KUKA KRL program: EPS_2_251806_MH56A_A_20260213065153.src

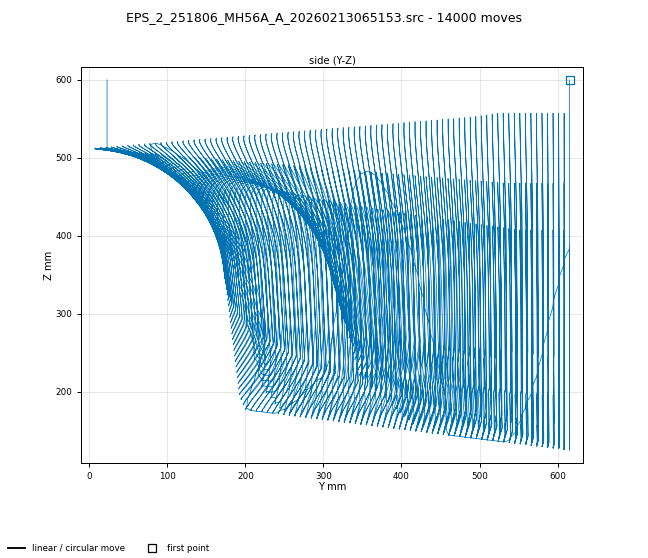
[picture p0: tool path of EPS_2_251806_MH56A_A_20260213065153.src, 14000 of 14002 moves have a stored position in this frame; points joined in program order, loops and branches not executed]
&ACCESS RVP
&REL 4
&COMMENT QRS 19112012
&PARAM EDITMASK = *
DEF PART()
EXT BAS (BAS_COMMAND :IN,REAL :IN )
INT I
BAS (#INITMOV,0 )

;KUKA QRS Post kuka4.cps  Date:22-06-2017 !

File_ID=3030

QRS_PRE_INIT()

;Init var - Until changes are made in qrs_pre_init
Outlet_Square_prg=0
Inlet_1_Square_prg=0
Inlet_2_Square_prg=0
Inlet_3_Square_prg=0
Inlet_4_Square_prg=0
Inlet_5_Square_prg=0

Outlet_1={X 0.000, Y 529.100, Z 408.000, B 0.000, E1 0.000 }
Inlet_1={X 0.000, Y 549.850, Z 257.000, B 0.000, E1 90.000 }
Inlet_2={X 0.000, Y 535.660, Z 318.000, B 0.000, E1 180.000 }
Outlet_1_type=299
Inlet_1_type=201
Inlet_2_type=299
;QRS#1=Sidecore dimensions
;QRS#2=300-12" PVC SDR 35
;QRS#3=200-8" PVC SDR 35
;QRS#4=300-12" PVC SDR 35
;QRS#5=
;QRS#6=
;QRS#7=
;QRS#8=
;QRS#9=16M PSX
;QRS#10=12-08 PSX
;QRS#11=16M PSX
;QRS#12=
;QRS#13=
;QRS#14=
;QRS#15=
;QRS#16=1220x127x838 2,75'
;QRS#17=EPS Height
;QRS#18=557,5
;QRS#19=*
;QRS#20= UPDATED VERSION 22-06-2017
;QRS#21=*
Outlet_Square=0150
Inlet_1_Square=0100
Inlet_2_Square=0150
Inlet_3_Square=0
Inlet_4_Square=0
Inlet_5_Square=0
Mill_Square=1
Outlet_Square_Prg=206
Inlet_1_Square_prg=204
Inlet_2_Square_prg=206

QRS_INIT()

$ADVANCE=5

; T1
PTP {E1 173.498,E2 173.498}
PTP {X 0,Y 615.498,A -85,B 0,C 180,E1 173.498,E2 173.498,E3 0,E4 0,E5 0,E6 0}
QRS_SPEED_INIT()
LIN {X 0,Y 615.498,Z 600,A -85,B 0,C 180,E1 173.498,E2 173.498,E3 0,E4 0,E5 0,E6 0} C_VEL
LIN {X 0,Y 615.498,Z 398.232,A -85,B 0,C 180,E1 173.498,E2 173.498} C_VEL
LIN {X 0,Y 615.498,Z 387.353,A -85,B 0,C 180,E1 173.498,E2 173.498} C_VEL
LIN {X 0,Y 615.496,Z 385.709,A -85,B 0,C 180,E1 173.418,E2 173.418} C_VEL
LIN {X 0,Y 615.498,Z 378.036,A -85,B 0,C 180,E1 172.455,E2 172.455} C_VEL
LIN {X 0,Y 615.498,Z 368.258,A -85,B 0,C 180,E1 171.463,E2 171.463} C_VEL
LIN {X 0,Y 615.497,Z 357.992,A -85,B 0,C 180,E1 170.636,E2 170.636} C_VEL
LIN {X 0,Y 615.487,Z 346.429,A -85,B 0,C 180,E1 169.889,E2 169.889} C_VEL
LIN {X 0,Y 615.498,Z 334.597,A -85,B 0,C 180,E1 169.294,E2 169.294} C_VEL
LIN {X 0,Y 615.462,Z 321.661,A -85,B 0,C 180,E1 168.806,E2 168.806} C_VEL
LIN {X 0,Y 615.456,Z 309.061,A -85,B 0,C 180,E1 168.473,E2 168.473} C_VEL
LIN {X 0,Y 615.464,Z 295.936,A -85,B 0,C 180,E1 168.264,E2 168.264} C_VEL
LIN {X 0,Y 615.464,Z 195.1,A -85,B 0,C 180,E1 167.071,E2 167.071} C_VEL
LIN {X 0,Y 615.457,Z 175.283,A -85,B 0,C 180,E1 164.434,E2 164.434} C_VEL
LIN {X 0,Y 615.488,Z 153.929,A -85,B 0,C 180,E1 161.558,E2 161.558} C_VEL
LIN {X 0,Y 615.464,Z 133.353,A -85,B 0,C 180,E1 158.743,E2 158.743} C_VEL
LIN {X 0,Y 615.471,Z 125.313,A -85,B 0,C 180,E1 157.627,E2 157.627} C_VEL
LIN {X 0,Y 615.452,Z 125.319,A -85,B 0,C 180,E1 155.007,E2 155.007} C_VEL
LIN {X 0,Y 615.489,Z 125.315,A -85,B 0,C 180,E1 152.085,E2 152.085} C_VEL
LIN {X 0,Y 615.481,Z 125.311,A -85,B 0,C 180,E1 149.839,E2 149.839} C_VEL
LIN {X 0,Y 615.458,Z 125.315,A -85,B 0,C 180,E1 147.541,E2 147.541} C_VEL
LIN {X 0,Y 615.459,Z 125.319,A -85,B 0,C 180,E1 145.183,E2 145.183} C_VEL
LIN {X 0,Y 615.488,Z 125.327,A -85,B 0,C 180,E1 142.758,E2 142.758} C_VEL
LIN {X 0,Y 615.475,Z 125.311,A -85,B 0,C 180,E1 139.913,E2 139.913} C_VEL
LIN {X 0,Y 615.461,Z 125.315,A -85,B 0,C 180,E1 137.645,E2 137.645} C_VEL
LIN {X 0,Y 615.495,Z 125.326,A -85,B 0,C 180,E1 134.932,E2 134.932} C_VEL
LIN {X 0,Y 615.479,Z 125.31,A -85,B 0,C 180,E1 132.079,E2 132.079} C_VEL
LIN {X 0,Y 615.464,Z 125.315,A -85,B 0,C 180,E1 129.753,E2 129.753} C_VEL
LIN {X 0,Y 615.487,Z 125.321,A -85,B 0,C 180,E1 126.936,E2 126.936} C_VEL
LIN {X 0,Y 615.469,Z 125.313,A -85,B 0,C 180,E1 124.024,E2 124.024} C_VEL
LIN {X 0,Y 615.468,Z 125.319,A -85,B 0,C 180,E1 121.687,E2 121.687} C_VEL
LIN {X 0,Y 615.486,Z 125.326,A -85,B 0,C 180,E1 119.407,E2 119.407} C_VEL
LIN {X 0,Y 615.485,Z 125.308,A -85,B 0,C 180,E1 116.445,E2 116.445} C_VEL
LIN {X 0,Y 615.485,Z 125.326,A -85,B 0,C 180,E1 113.557,E2 113.557} C_VEL
LIN {X 0,Y 615.476,Z 125.335,A -85,B 0,C 180,E1 112.266,E2 112.266} C_VEL
LIN {X 0,Y 615.46,Z 145.204,A -85,B 0,C 180,E1 109.687,E2 109.687} C_VEL
LIN {X 0,Y 615.464,Z 157.175,A -85,B 0,C 180,E1 108.18,E2 108.18} C_VEL
LIN {X 0,Y 615.492,Z 321.221,A -85,B 0,C 180,E1 106.201,E2 106.201} C_VEL
LIN {X 0,Y 615.489,Z 335.787,A -85,B 0,C 180,E1 105.906,E2 105.906} C_VEL
LIN {X 0,Y 615.477,Z 350.397,A -85,B 0,C 180,E1 105.481,E2 105.481} C_VEL
LIN {X 0,Y 615.492,Z 363.722,A -85,B 0,C 180,E1 104.973,E2 104.973} C_VEL
LIN {X 0,Y 615.483,Z 377.372,A -85,B 0,C 180,E1 104.32,E2 104.32} C_VEL
LIN {X 0,Y 615.5,Z 390.656,A -85,B 0,C 180,E1 103.538,E2 103.538} C_VEL
LIN {X 0,Y 615.497,Z 402.508,A -85,B 0,C 180,E1 102.698,E2 102.698} C_VEL
LIN {X 0,Y 615.497,Z 414.352,A -85,B 0,C 180,E1 101.694,E2 101.694} C_VEL
LIN {X 0,Y 615.495,Z 424.163,A -85,B 0,C 180,E1 100.709,E2 100.709} C_VEL
LIN {X 0,Y 615.495,Z 434.007,A -85,B 0,C 180,E1 99.531,E2 99.531} C_VEL
LIN {X 0,Y 615.497,Z 442.098,A -85,B 0,C 180,E1 98.372,E2 98.372} C_VEL
LIN {X 0,Y 615.491,Z 448.779,A -85,B 0,C 180,E1 97.216,E2 97.216} C_VEL
LIN {X 0,Y 615.499,Z 454.945,A -85,B 0,C 180,E1 95.899,E2 95.899} C_VEL
LIN {X 0,Y 615.489,Z 459.714,A -85,B 0,C 180,E1 94.585,E2 94.585} C_VEL
LIN {X 0,Y 615.491,Z 463.219,A -85,B 0,C 180,E1 93.274,E2 93.274} C_VEL
LIN {X 0,Y 615.5,Z 465.539,A -85,B 0,C 180,E1 91.964,E2 91.964} C_VEL
LIN {X 0,Y 615.491,Z 466.728,A -85,B 0,C 180,E1 90.655,E2 90.655} C_VEL
LIN {X 0,Y 615.492,Z 466.751,A -85,B 0,C 180,E1 89.347,E2 89.347} C_VEL
LIN {X 0,Y 615.5,Z 465.647,A -85,B 0,C 180,E1 88.038,E2 88.038} C_VEL
LIN {X 0,Y 615.494,Z 463.417,A -85,B 0,C 180,E1 86.728,E2 86.728} C_VEL
LIN {X 0,Y 615.49,Z 460.008,A -85,B 0,C 180,E1 85.416,E2 85.416} C_VEL
LIN {X 0,Y 615.499,Z 455.339,A -85,B 0,C 180,E1 84.102,E2 84.102} C_VEL
LIN {X 0,Y 615.491,Z 449.277,A -85,B 0,C 180,E1 82.785,E2 82.785} C_VEL
LIN {X 0,Y 615.493,Z 441.639,A -85,B 0,C 180,E1 81.464,E2 81.464} C_VEL
LIN {X 0,Y 615.496,Z 433.457,A -85,B 0,C 180,E1 80.305,E2 80.305} C_VEL
LIN {X 0,Y 615.495,Z 423.338,A -85,B 0,C 180,E1 79.109,E2 79.109} C_VEL
LIN {X 0,Y 615.497,Z 411.693,A -85,B 0,C 180,E1 77.973,E2 77.973} C_VEL
LIN {X 0,Y 615.498,Z 400.425,A -85,B 0,C 180,E1 77.052,E2 77.052} C_VEL
LIN {X 0,Y 615.498,Z 388.189,A -85,B 0,C 180,E1 76.211,E2 76.211} C_VEL
LIN {X 0,Y 615.49,Z 374.794,A -85,B 0,C 180,E1 75.452,E2 75.452} C_VEL
LIN {X 0,Y 615.488,Z 359.885,A -85,B 0,C 180,E1 74.775,E2 74.775} C_VEL
LIN {X 0,Y 615.476,Z 345.415,A -85,B 0,C 180,E1 74.266,E2 74.266} C_VEL
LIN {X 0,Y 615.492,Z 329.776,A -85,B 0,C 180,E1 73.865,E2 73.865} C_VEL
LIN {X 0,Y 615.492,Z 314.76,A -85,B 0,C 180,E1 73.618,E2 73.618} C_VEL
LIN {X 0,Y 615.47,Z 156.862,A -85,B 0,C 180,E1 71.72,E2 71.72} C_VEL
LIN {X 0,Y 615.478,Z 135.121,A -85,B 0,C 180,E1 68.92,E2 68.92} C_VEL
LIN {X 0,Y 615.483,Z 125.31,A -85,B 0,C 180,E1 67.625,E2 67.625} C_VEL
LIN {X 0,Y 615.478,Z 125.313,A -85,B 0,C 180,E1 65.009,E2 65.009} C_VEL
LIN {X 0,Y 615.476,Z 125.318,A -85,B 0,C 180,E1 62.823,E2 62.823} C_VEL
LIN {X 0,Y 615.482,Z 125.319,A -85,B 0,C 180,E1 60.207,E2 60.207} C_VEL
LIN {X 0,Y 615.493,Z 125.306,A -85,B 0,C 180,E1 57.544,E2 57.544} C_VEL
LIN {X 0,Y 615.477,Z 125.312,A -85,B 0,C 180,E1 55.186,E2 55.186} C_VEL
LIN {X 0,Y 615.486,Z 125.322,A -85,B 0,C 180,E1 52.759,E2 52.759} C_VEL
LIN {X 0,Y 615.482,Z 125.31,A -85,B 0,C 180,E1 49.912,E2 49.912} C_VEL
LIN {X 0,Y 615.495,Z 125.306,A -85,B 0,C 180,E1 47.649,E2 47.649} C_VEL
LIN {X 0,Y 615.478,Z 125.321,A -85,B 0,C 180,E1 44.932,E2 44.932} C_VEL
LIN {X 0,Y 615.483,Z 125.311,A -85,B 0,C 180,E1 42.082,E2 42.082} C_VEL
LIN {X 0,Y 615.489,Z 125.307,A -85,B 0,C 180,E1 39.75,E2 39.75} C_VEL
LIN {X 0,Y 615.482,Z 125.324,A -85,B 0,C 180,E1 36.938,E2 36.938} C_VEL
LIN {X 0,Y 615.488,Z 125.308,A -85,B 0,C 180,E1 34.022,E2 34.022} C_VEL
LIN {X 0,Y 615.479,Z 125.322,A -85,B 0,C 180,E1 31.087,E2 31.087} C_VEL
LIN {X 0,Y 615.482,Z 125.314,A -85,B 0,C 180,E1 28.452,E2 28.452} C_VEL
LIN {X 0,Y 615.476,Z 125.311,A -85,B 0,C 180,E1 25.716,E2 25.716} C_VEL
LIN {X 0,Y 615.472,Z 125.315,A -85,B 0,C 180,E1 23.557,E2 23.557} C_VEL
LIN {X 0,Y 615.473,Z 125.318,A -85,B 0,C 180,E1 21.433,E2 21.433} C_VEL
LIN {X 0,Y 615.483,Z 125.315,A -85,B 0,C 180,E1 18.608,E2 18.608} C_VEL
LIN {X 0,Y 615.476,Z 125.311,A -85,B 0,C 180,E1 15.906,E2 15.906} C_VEL
LIN {X 0,Y 615.49,Z 125.325,A -85,B 0,C 180,E1 13.201,E2 13.201} C_VEL
LIN {X 0,Y 615.488,Z 125.31,A -85,B 0,C 180,E1 10.527,E2 10.527} C_VEL
LIN {X 0,Y 615.47,Z 125.313,A -85,B 0,C 180,E1 7.876,E2 7.876} C_VEL
LIN {X 0,Y 615.493,Z 125.327,A -85,B 0,C 180,E1 5.241,E2 5.241} C_VEL
LIN {X 0,Y 615.491,Z 125.309,A -85,B 0,C 180,E1 2.618,E2 2.618} C_VEL
LIN {X 0,Y 615.469,Z 125.314,A -85,B 0,C 180,E1 0,E2 0} C_VEL
LIN {X 0,Y 615.489,Z 125.326,A -85,B 0,C 180,E1 -2.618,E2 -2.618} C_VEL
LIN {X 0,Y 615.491,Z 125.31,A -85,B 0,C 180,E1 -5.241,E2 -5.241} C_VEL
LIN {X 0,Y 615.467,Z 125.314,A -85,B 0,C 180,E1 -7.876,E2 -7.876} C_VEL
LIN {X 0,Y 615.489,Z 125.327,A -85,B 0,C 180,E1 -10.527,E2 -10.527} C_VEL
LIN {X 0,Y 615.495,Z 125.308,A -85,B 0,C 180,E1 -13.201,E2 -13.201} C_VEL
LIN {X 0,Y 615.465,Z 125.316,A -85,B 0,C 180,E1 -15.906,E2 -15.906} C_VEL
LIN {X 0,Y 615.49,Z 125.32,A -85,B 0,C 180,E1 -18.646,E2 -18.646} C_VEL
LIN {X 0,Y 615.475,Z 125.31,A -85,B 0,C 180,E1 -21.432,E2 -21.432} C_VEL
LIN {X 0,Y 615.486,Z 125.325,A -85,B 0,C 180,E1 -24.272,E2 -24.272} C_VEL
LIN {X 0,Y 615.487,Z 125.308,A -85,B 0,C 180,E1 -27.177,E2 -27.177} C_VEL
LIN {X 0,Y 615.465,Z 125.318,A -85,B 0,C 180,E1 -29.793,E2 -29.793} C_VEL
LIN {X 0,Y 615.49,Z 125.32,A -85,B 0,C 180,E1 -32.457,E2 -32.457} C_VEL
LIN {X 0,Y 615.493,Z 125.309,A -85,B 0,C 180,E1 -34.815,E2 -34.815} C_VEL
LIN {X 0,Y 615.469,Z 125.312,A -85,B 0,C 180,E1 -37.243,E2 -37.243} C_VEL
LIN {X 0,Y 615.494,Z 125.324,A -85,B 0,C 180,E1 -40.092,E2 -40.092} C_VEL
LIN {X 0,Y 615.474,Z 125.31,A -85,B 0,C 180,E1 -43.048,E2 -43.048} C_VEL
LIN {X 0,Y 615.478,Z 125.322,A -85,B 0,C 180,E1 -45.851,E2 -45.851} C_VEL
LIN {X 0,Y 615.493,Z 125.311,A -85,B 0,C 180,E1 -48.528,E2 -48.528} C_VEL
LIN {X 0,Y 615.464,Z 125.313,A -85,B 0,C 180,E1 -51.095,E2 -51.095} C_VEL
LIN {X 0,Y 615.466,Z 125.32,A -85,B 0,C 180,E1 -53.575,E2 -53.575} C_VEL
LIN {X 0,Y 615.495,Z 125.31,A -85,B 0,C 180,E1 -56.465,E2 -56.465} C_VEL
LIN {X 0,Y 615.459,Z 125.315,A -85,B 0,C 180,E1 -59.08,E2 -59.08} C_VEL
LIN {X 0,Y 615.471,Z 125.321,A -85,B 0,C 180,E1 -61.553,E2 -61.553} C_VEL
LIN {X 0,Y 615.473,Z 125.335,A -85,B 0,C 180,E1 -62.731,E2 -62.731} C_VEL
LIN {X 0,Y 615.474,Z 159.072,A -85,B 0,C 180,E1 -65.369,E2 -65.369} C_VEL
LIN {X 0,Y 615.491,Z 196.299,A -85,B 0,C 180,E1 -68.218,E2 -68.218} C_VEL
LIN {X 0,Y 615.474,Z 234.689,A -85,B 0,C 180,E1 -71.095,E2 -71.095} C_VEL
LIN {X 0,Y 615.483,Z 243.095,A -85,B 0,C 180,E1 -71.719,E2 -71.719} C_VEL
LIN {X 0,Y 615.482,Z 412.295,A -85,B 0,C 180,E1 -73.77,E2 -73.77} C_VEL
LIN {X 0,Y 615.496,Z 427.753,A -85,B 0,C 180,E1 -74.096,E2 -74.096} C_VEL
LIN {X 0,Y 615.481,Z 443.079,A -85,B 0,C 180,E1 -74.563,E2 -74.563} C_VEL
LIN {X 0,Y 615.497,Z 456.777,A -85,B 0,C 180,E1 -75.114,E2 -75.114} C_VEL
LIN {X 0,Y 615.495,Z 471.053,A -85,B 0,C 180,E1 -75.834,E2 -75.834} C_VEL
LIN {X 0,Y 615.497,Z 483.914,A -85,B 0,C 180,E1 -76.632,E2 -76.632} C_VEL
LIN {X 0,Y 615.495,Z 496.267,A -85,B 0,C 180,E1 -77.555,E2 -77.555} C_VEL
LIN {X 0,Y 615.495,Z 506.617,A -85,B 0,C 180,E1 -78.474,E2 -78.474} C_VEL
LIN {X 0,Y 615.495,Z 516.193,A -85,B 0,C 180,E1 -79.474,E2 -79.474} C_VEL
LIN {X 0,Y 615.493,Z 525.584,A -85,B 0,C 180,E1 -80.637,E2 -80.637} C_VEL
LIN {X 0,Y 615.494,Z 533.386,A -85,B 0,C 180,E1 -81.795,E2 -81.795} C_VEL
LIN {X 0,Y 615.496,Z 540.608,A -85,B 0,C 180,E1 -83.102,E2 -83.102} C_VEL
LIN {X 0,Y 615.499,Z 546.44,A -85,B 0,C 180,E1 -84.431,E2 -84.431} C_VEL
LIN {X 0,Y 615.491,Z 549.863,A -85,B 0,C 180,E1 -85.416,E2 -85.416} C_VEL
LIN {X 0,Y 615.492,Z 553.32,A -85,B 0,C 180,E1 -86.728,E2 -86.728} C_VEL
LIN {X 0,Y 615.499,Z 555.594,A -85,B 0,C 180,E1 -88.038,E2 -88.038} C_VEL
LIN {X 0,Y 615.494,Z 556.741,A -85,B 0,C 180,E1 -89.347,E2 -89.347} C_VEL
LIN {X 0,Y 615.494,Z 556.74,A -85,B 0,C 180,E1 -90.655,E2 -90.655} C_VEL
LIN {X 0,Y 615.499,Z 555.592,A -85,B 0,C 180,E1 -91.964,E2 -91.964} C_VEL
LIN {X 0,Y 615.492,Z 553.316,A -85,B 0,C 180,E1 -93.274,E2 -93.274} C_VEL
LIN {X 0,Y 615.491,Z 549.858,A -85,B 0,C 180,E1 -94.585,E2 -94.585} C_VEL
LIN {X 0,Y 615.499,Z 545.138,A -85,B 0,C 180,E1 -95.899,E2 -95.899} C_VEL
LIN {X 0,Y 615.494,Z 539.025,A -85,B 0,C 180,E1 -97.216,E2 -97.216} C_VEL
LIN {X 0,Y 615.494,Z 531.327,A -85,B 0,C 180,E1 -98.537,E2 -98.537} C_VEL
LIN {X 0,Y 615.495,Z 523.108,A -85,B 0,C 180,E1 -99.697,E2 -99.697} C_VEL
LIN {X 0,Y 615.497,Z 512.892,A -85,B 0,C 180,E1 -100.893,E2 -100.893} C_VEL
LIN {X 0,Y 615.495,Z 503.059,A -85,B 0,C 180,E1 -101.861,E2 -101.861} C_VEL
LIN {X 0,Y 615.497,Z 490.937,A -85,B 0,C 180,E1 -102.866,E2 -102.866} C_VEL
LIN {X 0,Y 615.498,Z 478.786,A -85,B 0,C 180,E1 -103.706,E2 -103.706} C_VEL
LIN {X 0,Y 615.488,Z 465.367,A -85,B 0,C 180,E1 -104.473,E2 -104.473} C_VEL
LIN {X 0,Y 615.497,Z 450.831,A -85,B 0,C 180,E1 -105.142,E2 -105.142} C_VEL
LIN {X 0,Y 615.495,Z 436.593,A -85,B 0,C 180,E1 -105.651,E2 -105.651} C_VEL
LIN {X 0,Y 615.498,Z 422.148,A -85,B 0,C 180,E1 -106.035,E2 -106.035} C_VEL
LIN {X 0,Y 615.479,Z 407.742,A -85,B 0,C 180,E1 -106.296,E2 -106.296} C_VEL
LIN {X 0,Y 615.483,Z 243.081,A -85,B 0,C 180,E1 -108.282,E2 -108.282} C_VEL
LIN {X 0,Y 615.495,Z 205.582,A -85,B 0,C 180,E1 -111.081,E2 -111.081} C_VEL
LIN {X 0,Y 615.487,Z 170.098,A -85,B 0,C 180,E1 -113.78,E2 -113.78} C_VEL
LIN {X 0,Y 615.473,Z 135.781,A -85,B 0,C 180,E1 -116.445,E2 -116.445} C_VEL
LIN {X 0,Y 615.47,Z 125.313,A -85,B 0,C 180,E1 -117.271,E2 -117.271} C_VEL
LIN {X 0,Y 615.483,Z 125.324,A -85,B 0,C 180,E1 -120.161,E2 -120.161} C_VEL
LIN {X 0,Y 615.45,Z 125.321,A -85,B 0,C 180,E1 -122.46,E2 -122.46} C_VEL
LIN {X 0,Y 615.447,Z 125.318,A -85,B 0,C 180,E1 -124.818,E2 -124.818} C_VEL
LIN {X 0,Y 615.477,Z 125.316,A -85,B 0,C 180,E1 -127.244,E2 -127.244} C_VEL
LIN {X 0,Y 615.446,Z 125.323,A -85,B 0,C 180,E1 -130.085,E2 -130.085} C_VEL
LIN {X 0,Y 615.43,Z 125.322,A -85,B 0,C 180,E1 -132.359,E2 -132.359} C_VEL
LIN {X 0,Y 615.457,Z 125.321,A -85,B 0,C 180,E1 -134.929,E2 -134.929} C_VEL
LIN {X 0,Y 615.451,Z 125.325,A -85,B 0,C 180,E1 -137.644,E2 -137.644} C_VEL
LIN {X 0,Y 615.415,Z 125.325,A -85,B 0,C 180,E1 -140.244,E2 -140.244} C_VEL
LIN {X 0,Y 615.455,Z 125.325,A -85,B 0,C 180,E1 -142.756,E2 -142.756} C_VEL
LIN {X 0,Y 615.468,Z 125.321,A -85,B 0,C 180,E1 -145.303,E2 -145.303} C_VEL
LIN {X 0,Y 615.432,Z 125.322,A -85,B 0,C 180,E1 -147.678,E2 -147.678} C_VEL
LIN {X 0,Y 615.431,Z 125.321,A -85,B 0,C 180,E1 -149.837,E2 -149.837} C_VEL
LIN {X 0,Y 615.441,Z 125.322,A -85,B 0,C 180,E1 -152.083,E2 -152.083} C_VEL
LIN {X 0,Y 615.477,Z 125.325,A -85,B 0,C 180,E1 -154.434,E2 -154.434} C_VEL
LIN {X 0,Y 615.469,Z 125.315,A -85,B 0,C 180,E1 -157.155,E2 -157.155} C_VEL
LIN {X 0,Y 615.446,Z 125.455,A -85,B 0,C 180,E1 -157.739,E2 -157.739} C_VEL
LIN {X 0,Y 615.475,Z 144.141,A -85,B 0,C 180,E1 -160.315,E2 -160.315} C_VEL
LIN {X 0,Y 615.474,Z 165.728,A -85,B 0,C 180,E1 -163.242,E2 -163.242} C_VEL
LIN {X 0,Y 615.456,Z 185.766,A -85,B 0,C 180,E1 -165.922,E2 -165.922} C_VEL
LIN {X 0,Y 615.467,Z 195.354,A -85,B 0,C 180,E1 -167.176,E2 -167.176} C_VEL
LIN {X 0,Y 615.489,Z 303.148,A -85,B 0,C 180,E1 -168.452,E2 -168.452} C_VEL
LIN {X 0,Y 615.494,Z 315.725,A -85,B 0,C 180,E1 -168.724,E2 -168.724} C_VEL
LIN {X 0,Y 615.493,Z 329.078,A -85,B 0,C 180,E1 -169.157,E2 -169.157} C_VEL
LIN {X 0,Y 615.47,Z 340.07,A -85,B 0,C 180,E1 -169.639,E2 -169.639} C_VEL
LIN {X 0,Y 615.47,Z 351.809,A -85,B 0,C 180,E1 -170.304,E2 -170.304} C_VEL
LIN {X 0,Y 615.499,Z 362.268,A -85,B 0,C 180,E1 -171.05,E2 -171.05} C_VEL
LIN {X 0,Y 615.498,Z 370.831,A -85,B 0,C 180,E1 -171.794,E2 -171.794} C_VEL
LIN {X 0,Y 615.497,Z 378.71,A -85,B 0,C 180,E1 -172.62,E2 -172.62} C_VEL
LIN {X 0,Y 615.497,Z 386.399,A -85,B 0,C 180,E1 -173.608,E2 -173.608} C_VEL
LIN {X 0,Y 615.497,Z 393.458,A -85,B 0,C 180,E1 -174.759,E2 -174.759} C_VEL
LIN {X 0,Y 615.497,Z 398.157,A -85,B 0,C 180,E1 -175.744,E2 -175.744} C_VEL
LIN {X 0,Y 615.495,Z 401.755,A -85,B 0,C 180,E1 -176.727,E2 -176.727} C_VEL
LIN {X 0,Y 615.496,Z 403.615,A -85,B 0,C 180,E1 -177.382,E2 -177.382} C_VEL
LIN {X 0,Y 615.497,Z 405.034,A -85,B 0,C 180,E1 -178.037,E2 -178.037} C_VEL
LIN {X 0,Y 615.497,Z 406.641,A -85,B 0,C 180,E1 -179.346,E2 -179.346} C_VEL
LIN {X 0,Y 615.494,Z 406.884,A -85,B 0,C 180,E1 -180,E2 -180} C_VEL
LIN {X 0,Y 615.495,Z 406.705,A -85,B 0,C 180,E1 -180.654,E2 -180.654} C_VEL
LIN {X 0,Y 615.496,Z 405.183,A -85,B 0,C 180,E1 -181.963,E2 -181.963} C_VEL
LIN {X 0,Y 615.498,Z 403.841,A -85,B 0,C 180,E1 -182.618,E2 -182.618} C_VEL
LIN {X 0,Y 615.497,Z 400.994,A -85,B 0,C 180,E1 -183.601,E2 -183.601} C_VEL
LIN {X 0,Y 615.498,Z 397.134,A -85,B 0,C 180,E1 -184.585,E2 -184.585} C_VEL
LIN {X 0,Y 615.498,Z 392.151,A -85,B 0,C 180,E1 -185.57,E2 -185.57} C_VEL
LIN {X 0,Y 615.496,Z 385.709,A -85,B 0,C 180,E1 -186.582,E2 -186.582} C_VEL
LIN {X 0,Y 614.829,Z 382.527,A -85,B 0,C 180,E1 -187.031,E2 -187.031} C_VEL
LIN {X 0,Y 611.989,Z 376.954,A -85,B 0,C 180,E1 -187.748,E2 -187.748} C_VEL
LIN {X 0,Y 609.138,Z 370.679,A -85,B 0,C 180,E1 -188.429,E2 -188.429} C_VEL
LIN {X 0,Y 608.477,Z 366.438,A -85,B 0,C 180,E1 -188.819,E2 -188.819} C_VEL
LIN {X 0,Y 608.491,Z 355.888,A -85,B 0,C 180,E1 -189.641,E2 -189.641} C_VEL
LIN {X 0,Y 608.492,Z 345.11,A -85,B 0,C 180,E1 -190.313,E2 -190.313} C_VEL
LIN {X 0,Y 608.518,Z 332.676,A -85,B 0,C 180,E1 -190.918,E2 -190.918} C_VEL
LIN {X 0,Y 608.496,Z 320.463,A -85,B 0,C 180,E1 -191.366,E2 -191.366} C_VEL
LIN {X 0,Y 608.528,Z 308.153,A -85,B 0,C 180,E1 -191.682,E2 -191.682} C_VEL
LIN {X 0,Y 608.54,Z 294.245,A -85,B 0,C 180,E1 -191.893,E2 -191.893} C_VEL
LIN {X 0,Y 608.511,Z 195.849,A -85,B 0,C 180,E1 -193.058,E2 -193.058} C_VEL
LIN {X 0,Y 608.45,Z 195.084,A -85,B 0,C 180,E1 -193.102,E2 -193.102} C_VEL
LIN {X 0,Y 608.469,Z 176.629,A -85,B 0,C 180,E1 -195.578,E2 -195.578} C_VEL
LIN {X 0,Y 608.533,Z 155.148,A -85,B 0,C 180,E1 -198.496,E2 -198.496} C_VEL
LIN {X 0,Y 608.55,Z 134.625,A -85,B 0,C 180,E1 -201.333,E2 -201.333} C_VEL
LIN {X 0,Y 608.458,Z 126.314,A -85,B 0,C 180,E1 -202.527,E2 -202.527} C_VEL
LIN {X 0,Y 608.438,Z 126.315,A -85,B 0,C 180,E1 -204.572,E2 -204.572} C_VEL
LIN {X 0,Y 608.461,Z 126.317,A -85,B 0,C 180,E1 -207.203,E2 -207.203} C_VEL
LIN {X 0,Y 608.471,Z 126.313,A -85,B 0,C 180,E1 -209.971,E2 -209.971} C_VEL
LIN {X 0,Y 608.448,Z 126.316,A -85,B 0,C 180,E1 -212.88,E2 -212.88} C_VEL
LIN {X 0,Y 608.437,Z 126.325,A -85,B 0,C 180,E1 -215.278,E2 -215.278} C_VEL
LIN {X 0,Y 608.466,Z 126.314,A -85,B 0,C 180,E1 -217.747,E2 -217.747} C_VEL
LIN {X 0,Y 608.437,Z 126.315,A -85,B 0,C 180,E1 -220.327,E2 -220.327} C_VEL
LIN {X 0,Y 608.481,Z 126.316,A -85,B 0,C 180,E1 -223.309,E2 -223.309} C_VEL
LIN {X 0,Y 608.461,Z 126.312,A -85,B 0,C 180,E1 -226.129,E2 -226.129} C_VEL
LIN {X 0,Y 608.45,Z 126.321,A -85,B 0,C 180,E1 -228.822,E2 -228.822} C_VEL
LIN {X 0,Y 608.461,Z 126.312,A -85,B 0,C 180,E1 -231.761,E2 -231.761} C_VEL
LIN {X 0,Y 608.444,Z 126.314,A -85,B 0,C 180,E1 -233.955,E2 -233.955} C_VEL
LIN {X 0,Y 608.447,Z 126.317,A -85,B 0,C 180,E1 -236.328,E2 -236.328} C_VEL
LIN {X 0,Y 608.45,Z 126.324,A -85,B 0,C 180,E1 -238.732,E2 -238.732} C_VEL
LIN {X 0,Y 608.474,Z 126.311,A -85,B 0,C 180,E1 -241.38,E2 -241.38} C_VEL
LIN {X 0,Y 608.441,Z 126.316,A -85,B 0,C 180,E1 -243.964,E2 -243.964} C_VEL
LIN {X 0,Y 608.458,Z 126.317,A -85,B 0,C 180,E1 -246.154,E2 -246.154} C_VEL
LIN {X 0,Y 608.463,Z 126.324,A -85,B 0,C 180,E1 -247.594,E2 -247.594} C_VEL
LIN {X 0,Y 608.58,Z 142.516,A -85,B 0,C 180,E1 -249.729,E2 -249.729} C_VEL
LIN {X 0,Y 608.554,Z 157.221,A -85,B 0,C 180,E1 -251.606,E2 -251.606} C_VEL
LIN {X 0,Y 608.704,Z 288.325,A -85,B 0,C 180,E1 -253.201,E2 -253.201} C_VEL
LIN {X 0,Y 608.686,Z 323.244,A -85,B 0,C 180,E1 -253.646,E2 -253.646} C_VEL
LIN {X 0,Y 608.639,Z 339.157,A -85,B 0,C 180,E1 -253.996,E2 -253.996} C_VEL
LIN {X 0,Y 608.625,Z 354.105,A -85,B 0,C 180,E1 -254.469,E2 -254.469} C_VEL
LIN {X 0,Y 608.595,Z 367.638,A -85,B 0,C 180,E1 -255.025,E2 -255.025} C_VEL
LIN {X 0,Y 608.572,Z 381.425,A -85,B 0,C 180,E1 -255.734,E2 -255.734} C_VEL
LIN {X 0,Y 608.548,Z 394.536,A -85,B 0,C 180,E1 -256.56,E2 -256.56} C_VEL
LIN {X 0,Y 608.505,Z 406.826,A -85,B 0,C 180,E1 -257.492,E2 -257.492} C_VEL
LIN {X 0,Y 608.498,Z 418.038,A -85,B 0,C 180,E1 -258.507,E2 -258.507} C_VEL
LIN {X 0,Y 608.477,Z 428.926,A -85,B 0,C 180,E1 -259.686,E2 -259.686} C_VEL
LIN {X 0,Y 608.469,Z 437.973,A -85,B 0,C 180,E1 -260.861,E2 -260.861} C_VEL
LIN {X 0,Y 608.457,Z 445.474,A -85,B 0,C 180,E1 -262.032,E2 -262.032} C_VEL
LIN {X 0,Y 608.446,Z 452.626,A -85,B 0,C 180,E1 -263.396,E2 -263.396} C_VEL
LIN {X 0,Y 608.435,Z 457.992,A -85,B 0,C 180,E1 -264.697,E2 -264.697} C_VEL
LIN {X 0,Y 608.432,Z 462.164,A -85,B 0,C 180,E1 -266.025,E2 -266.025} C_VEL
LIN {X 0,Y 608.421,Z 465.108,A -85,B 0,C 180,E1 -267.351,E2 -267.351} C_VEL
LIN {X 0,Y 608.444,Z 466.881,A -85,B 0,C 180,E1 -268.675,E2 -268.675} C_VEL
LIN {X 0,Y 608.432,Z 467.495,A -85,B 0,C 180,E1 -269.999,E2 -269.999} C_VEL
LIN {X 0,Y 608.446,Z 466.945,A -85,B 0,C 180,E1 -271.323,E2 -271.323} C_VEL
LIN {X 0,Y 608.424,Z 465.261,A -85,B 0,C 180,E1 -272.647,E2 -272.647} C_VEL
LIN {X 0,Y 608.431,Z 462.409,A -85,B 0,C 180,E1 -273.973,E2 -273.973} C_VEL
LIN {X 0,Y 608.435,Z 458.333,A -85,B 0,C 180,E1 -275.301,E2 -275.301} C_VEL
LIN {X 0,Y 608.445,Z 452.927,A -85,B 0,C 180,E1 -276.632,E2 -276.632} C_VEL
LIN {X 0,Y 608.456,Z 446.026,A -85,B 0,C 180,E1 -277.966,E2 -277.966} C_VEL
LIN {X 0,Y 608.466,Z 438.598,A -85,B 0,C 180,E1 -279.137,E2 -279.137} C_VEL
LIN {X 0,Y 608.476,Z 429.667,A -85,B 0,C 180,E1 -280.312,E2 -280.312} C_VEL
LIN {X 0,Y 608.494,Z 418.959,A -85,B 0,C 180,E1 -281.491,E2 -281.491} C_VEL
LIN {X 0,Y 608.513,Z 406.91,A -85,B 0,C 180,E1 -282.59,E2 -282.59} C_VEL
LIN {X 0,Y 608.543,Z 394.635,A -85,B 0,C 180,E1 -283.524,E2 -283.524} C_VEL
LIN {X 0,Y 608.588,Z 381.692,A -85,B 0,C 180,E1 -284.341,E2 -284.341} C_VEL
LIN {X 0,Y 608.606,Z 367.774,A -85,B 0,C 180,E1 -285.059,E2 -285.059} C_VEL
LIN {X 0,Y 608.627,Z 353.109,A -85,B 0,C 180,E1 -285.658,E2 -285.658} C_VEL
LIN {X 0,Y 608.663,Z 337.56,A -85,B 0,C 180,E1 -286.137,E2 -286.137} C_VEL
LIN {X 0,Y 608.692,Z 322.143,A -85,B 0,C 180,E1 -286.463,E2 -286.463} C_VEL
LIN {X 0,Y 608.597,Z 157.486,A -85,B 0,C 180,E1 -288.479,E2 -288.479} C_VEL
LIN {X 0,Y 608.528,Z 156.879,A -85,B 0,C 180,E1 -288.496,E2 -288.496} C_VEL
LIN {X 0,Y 608.557,Z 136.468,A -85,B 0,C 180,E1 -291.154,E2 -291.154} C_VEL
LIN {X 0,Y 608.469,Z 126.312,A -85,B 0,C 180,E1 -292.505,E2 -292.505} C_VEL
LIN {X 0,Y 608.452,Z 126.319,A -85,B 0,C 180,E1 -295.3,E2 -295.3} C_VEL
LIN {X 0,Y 608.442,Z 126.324,A -85,B 0,C 180,E1 -297.517,E2 -297.517} C_VEL
LIN {X 0,Y 608.462,Z 126.315,A -85,B 0,C 180,E1 -299.97,E2 -299.97} C_VEL
LIN {X 0,Y 608.466,Z 126.311,A -85,B 0,C 180,E1 -302.523,E2 -302.523} C_VEL
LIN {X 0,Y 608.441,Z 126.322,A -85,B 0,C 180,E1 -305.276,E2 -305.276} C_VEL
LIN {X 0,Y 608.466,Z 126.316,A -85,B 0,C 180,E1 -307.745,E2 -307.745} C_VEL
LIN {X 0,Y 608.447,Z 126.313,A -85,B 0,C 180,E1 -310.328,E2 -310.328} C_VEL
LIN {X 0,Y 608.476,Z 126.32,A -85,B 0,C 180,E1 -313.309,E2 -313.309} C_VEL
LIN {X 0,Y 608.468,Z 126.311,A -85,B 0,C 180,E1 -316.13,E2 -316.13} C_VEL
LIN {X 0,Y 608.447,Z 126.317,A -85,B 0,C 180,E1 -318.823,E2 -318.823} C_VEL
LIN {X 0,Y 608.467,Z 126.318,A -85,B 0,C 180,E1 -321.412,E2 -321.412} C_VEL
LIN {X 0,Y 608.473,Z 126.31,A -85,B 0,C 180,E1 -323.949,E2 -323.949} C_VEL
LIN {X 0,Y 608.457,Z 126.312,A -85,B 0,C 180,E1 -326.329,E2 -326.329} C_VEL
LIN {X 0,Y 608.469,Z 126.314,A -85,B 0,C 180,E1 -328.727,E2 -328.727} C_VEL
LIN {X 0,Y 608.47,Z 126.316,A -85,B 0,C 180,E1 -331.378,E2 -331.378} C_VEL
LIN {X 0,Y 608.438,Z 126.314,A -85,B 0,C 180,E1 -333.964,E2 -333.964} C_VEL
LIN {X 0,Y 608.465,Z 126.311,A -85,B 0,C 180,E1 -336.155,E2 -336.155} C_VEL
LIN {X 0,Y 608.449,Z 126.323,A -85,B 0,C 180,E1 -339.018,E2 -339.018} C_VEL
LIN {X 0,Y 608.444,Z 126.313,A -85,B 0,C 180,E1 -341.828,E2 -341.828} C_VEL
LIN {X 0,Y 608.468,Z 126.316,A -85,B 0,C 180,E1 -344.594,E2 -344.594} C_VEL
LIN {X 0,Y 608.476,Z 126.313,A -85,B 0,C 180,E1 -347.323,E2 -347.323} C_VEL
LIN {X 0,Y 608.444,Z 126.314,A -85,B 0,C 180,E1 -350.022,E2 -350.022} C_VEL
LIN {X 0,Y 608.478,Z 126.318,A -85,B 0,C 180,E1 -352.701,E2 -352.701} C_VEL
LIN {X 0,Y 608.457,Z 126.313,A -85,B 0,C 180,E1 -355.362,E2 -355.362} C_VEL
LIN {X 0,Y 608.44,Z 126.315,A -85,B 0,C 180,E1 -358.014,E2 -358.014} C_VEL
LIN {X 0,Y 608.481,Z 126.319,A -85,B 0,C 180,E1 -360.662,E2 -360.662} C_VEL
LIN {X 0,Y 608.478,Z 126.31,A -85,B 0,C 180,E1 -363.311,E2 -363.311} C_VEL
LIN {X 0,Y 608.444,Z 126.315,A -85,B 0,C 180,E1 -365.967,E2 -365.967} C_VEL
LIN {X 0,Y 608.458,Z 126.321,A -85,B 0,C 180,E1 -368.636,E2 -368.636} C_VEL
LIN {X 0,Y 608.471,Z 126.31,A -85,B 0,C 180,E1 -371.324,E2 -371.324} C_VEL
LIN {X 0,Y 608.456,Z 126.315,A -85,B 0,C 180,E1 -374.038,E2 -374.038} C_VEL
LIN {X 0,Y 608.473,Z 126.315,A -85,B 0,C 180,E1 -376.783,E2 -376.783} C_VEL
LIN {X 0,Y 608.445,Z 126.313,A -85,B 0,C 180,E1 -379.571,E2 -379.571} C_VEL
LIN {X 0,Y 608.484,Z 126.317,A -85,B 0,C 180,E1 -382.485,E2 -382.485} C_VEL
LIN {X 0,Y 608.441,Z 126.314,A -85,B 0,C 180,E1 -385.301,E2 -385.301} C_VEL
LIN {X 0,Y 608.441,Z 126.314,A -85,B 0,C 180,E1 -387.518,E2 -387.518} C_VEL
LIN {X 0,Y 608.454,Z 126.317,A -85,B 0,C 180,E1 -389.972,E2 -389.972} C_VEL
LIN {X 0,Y 608.462,Z 126.317,A -85,B 0,C 180,E1 -392.525,E2 -392.525} C_VEL
LIN {X 0,Y 608.432,Z 126.315,A -85,B 0,C 180,E1 -395.278,E2 -395.278} C_VEL
LIN {X 0,Y 608.462,Z 126.315,A -85,B 0,C 180,E1 -397.747,E2 -397.747} C_VEL
LIN {X 0,Y 608.473,Z 126.317,A -85,B 0,C 180,E1 -400.333,E2 -400.333} C_VEL
LIN {X 0,Y 608.443,Z 126.314,A -85,B 0,C 180,E1 -402.961,E2 -402.961} C_VEL
LIN {X 0,Y 608.447,Z 126.318,A -85,B 0,C 180,E1 -405.737,E2 -405.737} C_VEL
LIN {X 0,Y 608.463,Z 126.32,A -85,B 0,C 180,E1 -407.94,E2 -407.94} C_VEL
LIN {X 0,Y 608.467,Z 126.311,A -85,B 0,C 180,E1 -410.703,E2 -410.703} C_VEL
LIN {X 0,Y 608.434,Z 126.315,A -85,B 0,C 180,E1 -413.085,E2 -413.085} C_VEL
LIN {X 0,Y 608.455,Z 126.316,A -85,B 0,C 180,E1 -415.531,E2 -415.531} C_VEL
LIN {X 0,Y 608.462,Z 126.322,A -85,B 0,C 180,E1 -417.907,E2 -417.907} C_VEL
LIN {X 0,Y 608.473,Z 126.315,A -85,B 0,C 180,E1 -420.222,E2 -420.222} C_VEL
LIN {X 0,Y 608.507,Z 126.498,A -85,B 0,C 180,E1 -422.486,E2 -422.486} C_VEL
LIN {X 0,Y 608.869,Z 129.214,A -85,B 0,C 180,E1 -422.721,E2 -422.721} C_VEL
LIN {X 0,Y 608.797,Z 161.398,A -85,B 0,C 180,E1 -425.263,E2 -425.263} C_VEL
LIN {X 0,Y 608.731,Z 198.625,A -85,B 0,C 180,E1 -428.141,E2 -428.141} C_VEL
LIN {X 0,Y 608.619,Z 234.689,A -85,B 0,C 180,E1 -430.874,E2 -430.874} C_VEL
LIN {X 0,Y 608.647,Z 243.349,A -85,B 0,C 180,E1 -431.517,E2 -431.517} C_VEL
LIN {X 0,Y 608.674,Z 412.294,A -85,B 0,C 180,E1 -433.583,E2 -433.583} C_VEL
LIN {X 0,Y 608.67,Z 427.751,A -85,B 0,C 180,E1 -433.913,E2 -433.913} C_VEL
LIN {X 0,Y 608.629,Z 443.077,A -85,B 0,C 180,E1 -434.385,E2 -434.385} C_VEL
LIN {X 0,Y 608.606,Z 456.78,A -85,B 0,C 180,E1 -434.941,E2 -434.941} C_VEL
LIN {X 0,Y 608.577,Z 470.255,A -85,B 0,C 180,E1 -435.625,E2 -435.625} C_VEL
LIN {X 0,Y 608.554,Z 482.679,A -85,B 0,C 180,E1 -436.391,E2 -436.391} C_VEL
LIN {X 0,Y 608.528,Z 495.295,A -85,B 0,C 180,E1 -437.325,E2 -437.325} C_VEL
LIN {X 0,Y 608.496,Z 506.758,A -85,B 0,C 180,E1 -438.34,E2 -438.34} C_VEL
LIN {X 0,Y 608.477,Z 516.397,A -85,B 0,C 180,E1 -439.351,E2 -439.351} C_VEL
LIN {X 0,Y 608.476,Z 525.861,A -85,B 0,C 180,E1 -440.528,E2 -440.528} C_VEL
LIN {X 0,Y 608.456,Z 533.735,A -85,B 0,C 180,E1 -441.699,E2 -441.699} C_VEL
LIN {X 0,Y 608.44,Z 541.092,A -85,B 0,C 180,E1 -443.035,E2 -443.035} C_VEL
LIN {X 0,Y 608.45,Z 546.927,A -85,B 0,C 180,E1 -444.366,E2 -444.366} C_VEL
LIN {X 0,Y 608.427,Z 550.385,A -85,B 0,C 180,E1 -445.363,E2 -445.363} C_VEL
LIN {X 0,Y 608.421,Z 553.887,A -85,B 0,C 180,E1 -446.69,E2 -446.69} C_VEL
LIN {X 0,Y 608.444,Z 556.192,A -85,B 0,C 180,E1 -448.015,E2 -448.015} C_VEL
LIN {X 0,Y 608.436,Z 557.351,A -85,B 0,C 180,E1 -449.339,E2 -449.339} C_VEL
LIN {X 0,Y 608.436,Z 557.35,A -85,B 0,C 180,E1 -450.663,E2 -450.663} C_VEL
LIN {X 0,Y 608.444,Z 556.19,A -85,B 0,C 180,E1 -451.987,E2 -451.987} C_VEL
LIN {X 0,Y 608.421,Z 553.884,A -85,B 0,C 180,E1 -453.312,E2 -453.312} C_VEL
LIN {X 0,Y 608.427,Z 550.38,A -85,B 0,C 180,E1 -454.639,E2 -454.639} C_VEL
LIN {X 0,Y 608.437,Z 545.604,A -85,B 0,C 180,E1 -455.968,E2 -455.968} C_VEL
LIN {X 0,Y 608.457,Z 539.421,A -85,B 0,C 180,E1 -457.3,E2 -457.3} C_VEL
LIN {X 0,Y 608.468,Z 531.648,A -85,B 0,C 180,E1 -458.637,E2 -458.637} C_VEL
LIN {X 0,Y 608.471,Z 523.364,A -85,B 0,C 180,E1 -459.81,E2 -459.81} C_VEL
LIN {X 0,Y 608.493,Z 512.644,A -85,B 0,C 180,E1 -461.064,E2 -461.064} C_VEL
LIN {X 0,Y 608.522,Z 501.266,A -85,B 0,C 180,E1 -462.168,E2 -462.168} C_VEL
LIN {X 0,Y 608.548,Z 489.844,A -85,B 0,C 180,E1 -463.1,E2 -463.1} C_VEL
LIN {X 0,Y 608.565,Z 477.435,A -85,B 0,C 180,E1 -463.951,E2 -463.951} C_VEL
LIN {X 0,Y 608.575,Z 463.844,A -85,B 0,C 180,E1 -464.719,E2 -464.719} C_VEL
LIN {X 0,Y 608.639,Z 449.772,A -85,B 0,C 180,E1 -465.359,E2 -465.359} C_VEL
LIN {X 0,Y 608.645,Z 435.277,A -85,B 0,C 180,E1 -465.874,E2 -465.874} C_VEL
LIN {X 0,Y 608.682,Z 420.044,A -85,B 0,C 180,E1 -466.269,E2 -466.269} C_VEL
LIN {X 0,Y 608.68,Z 404.248,A -85,B 0,C 180,E1 -466.532,E2 -466.532} C_VEL
LIN {X 0,Y 608.622,Z 243.261,A -85,B 0,C 180,E1 -468.485,E2 -468.485} C_VEL
LIN {X 0,Y 608.714,Z 206.745,A -85,B 0,C 180,E1 -471.239,E2 -471.239} C_VEL
LIN {X 0,Y 608.768,Z 169.12,A -85,B 0,C 180,E1 -474.135,E2 -474.135} C_VEL
LIN {X 0,Y 608.859,Z 135.781,A -85,B 0,C 180,E1 -476.755,E2 -476.755} C_VEL
LIN {X 0,Y 608.855,Z 127.857,A -85,B 0,C 180,E1 -477.388,E2 -477.388} C_VEL
LIN {X 0,Y 608.472,Z 126.315,A -85,B 0,C 180,E1 -477.541,E2 -477.541} C_VEL
LIN {X 0,Y 608.436,Z 126.317,A -85,B 0,C 180,E1 -480.547,E2 -480.547} C_VEL
LIN {X 0,Y 608.44,Z 126.315,A -85,B 0,C 180,E1 -482.881,E2 -482.881} C_VEL
LIN {X 0,Y 608.436,Z 126.318,A -85,B 0,C 180,E1 -485.279,E2 -485.279} C_VEL
LIN {X 0,Y 608.452,Z 126.323,A -85,B 0,C 180,E1 -487.748,E2 -487.748} C_VEL
LIN {X 0,Y 608.406,Z 126.32,A -85,B 0,C 180,E1 -490.324,E2 -490.324} C_VEL
LIN {X 0,Y 608.43,Z 126.318,A -85,B 0,C 180,E1 -492.963,E2 -492.963} C_VEL
LIN {X 0,Y 608.418,Z 126.321,A -85,B 0,C 180,E1 -495.741,E2 -495.741} C_VEL
LIN {X 0,Y 608.412,Z 126.319,A -85,B 0,C 180,E1 -497.935,E2 -497.935} C_VEL
LIN {X 0,Y 608.42,Z 126.32,A -85,B 0,C 180,E1 -500.709,E2 -500.709} C_VEL
LIN {X 0,Y 608.445,Z 126.324,A -85,B 0,C 180,E1 -503.084,E2 -503.084} C_VEL
LIN {X 0,Y 608.441,Z 126.316,A -85,B 0,C 180,E1 -505.529,E2 -505.529} C_VEL
LIN {X 0,Y 608.42,Z 126.317,A -85,B 0,C 180,E1 -507.903,E2 -507.903} C_VEL
LIN {X 0,Y 608.428,Z 126.318,A -85,B 0,C 180,E1 -510.218,E2 -510.218} C_VEL
LIN {X 0,Y 608.487,Z 126.317,A -85,B 0,C 180,E1 -512.792,E2 -512.792} C_VEL
LIN {X 0,Y 608.434,Z 126.316,A -85,B 0,C 180,E1 -515.428,E2 -515.428} C_VEL
LIN {X 0,Y 608.436,Z 126.349,A -85,B 0,C 180,E1 -517.593,E2 -517.593} C_VEL
LIN {X 0,Y 608.553,Z 140.48,A -85,B 0,C 180,E1 -519.572,E2 -519.572} C_VEL
LIN {X 0,Y 608.521,Z 159.424,A -85,B 0,C 180,E1 -522.178,E2 -522.178} C_VEL
LIN {X 0,Y 608.488,Z 181.052,A -85,B 0,C 180,E1 -525.109,E2 -525.109} C_VEL
LIN {X 0,Y 608.469,Z 195.433,A -85,B 0,C 180,E1 -527.026,E2 -527.026} C_VEL
LIN {X 0,Y 608.548,Z 303.298,A -85,B 0,C 180,E1 -528.319,E2 -528.319} C_VEL
LIN {X 0,Y 608.536,Z 316.618,A -85,B 0,C 180,E1 -528.614,E2 -528.614} C_VEL
LIN {X 0,Y 608.526,Z 329.892,A -85,B 0,C 180,E1 -529.056,E2 -529.056} C_VEL
LIN {X 0,Y 608.483,Z 341.87,A -85,B 0,C 180,E1 -529.603,E2 -529.603} C_VEL
LIN {X 0,Y 608.482,Z 353.291,A -85,B 0,C 180,E1 -530.275,E2 -530.275} C_VEL
LIN {X 0,Y 608.474,Z 363.585,A -85,B 0,C 180,E1 -531.029,E2 -531.029} C_VEL
LIN {X 0,Y 608.464,Z 372.85,A -85,B 0,C 180,E1 -531.866,E2 -531.866} C_VEL
LIN {X 0,Y 608.466,Z 381.824,A -85,B 0,C 180,E1 -532.867,E2 -532.867} C_VEL
LIN {X 0,Y 608.444,Z 389.056,A -85,B 0,C 180,E1 -533.867,E2 -533.867} C_VEL
LIN {X 0,Y 608.462,Z 393.935,A -85,B 0,C 180,E1 -534.698,E2 -534.698} C_VEL
LIN {X 0,Y 608.441,Z 398.678,A -85,B 0,C 180,E1 -535.694,E2 -535.694} C_VEL
LIN {X 0,Y 608.425,Z 402.312,A -85,B 0,C 180,E1 -536.689,E2 -536.689} C_VEL
LIN {X 0,Y 608.425,Z 404.191,A -85,B 0,C 180,E1 -537.352,E2 -537.352} C_VEL
LIN {X 0,Y 608.442,Z 405.627,A -85,B 0,C 180,E1 -538.014,E2 -538.014} C_VEL
LIN {X 0,Y 608.44,Z 407.252,A -85,B 0,C 180,E1 -539.338,E2 -539.338} C_VEL
LIN {X 0,Y 608.434,Z 407.495,A -85,B 0,C 180,E1 -540,E2 -540} C_VEL
LIN {X 0,Y 608.438,Z 407.315,A -85,B 0,C 180,E1 -540.662,E2 -540.662} C_VEL
LIN {X 0,Y 608.441,Z 405.776,A -85,B 0,C 180,E1 -541.986,E2 -541.986} C_VEL
LIN {X 0,Y 608.426,Z 404.418,A -85,B 0,C 180,E1 -542.648,E2 -542.648} C_VEL
LIN {X 0,Y 608.45,Z 401.542,A -85,B 0,C 180,E1 -543.642,E2 -543.642} C_VEL
LIN {X 0,Y 608.433,Z 397.642,A -85,B 0,C 180,E1 -544.638,E2 -544.638} C_VEL
LIN {X 0,Y 608.45,Z 392.612,A -85,B 0,C 180,E1 -545.634,E2 -545.634} C_VEL
LIN {X 0,Y 608.441,Z 386.294,A -85,B 0,C 180,E1 -546.633,E2 -546.633} C_VEL
LIN {X 0,Y 608.476,Z 378.378,A -85,B 0,C 180,E1 -547.633,E2 -547.633} C_VEL
LIN {X 0,Y 608.472,Z 368.535,A -85,B 0,C 180,E1 -548.636,E2 -548.636} C_VEL
LIN {X 0,Y 608.477,Z 366.438,A -85,B 0,C 180,E1 -548.819,E2 -548.819} C_VEL
LIN {X 0,Y 607.809,Z 362.104,A -85,B 0,C 180,E1 -549.189,E2 -549.189} C_VEL
LIN {X 0,Y 604.966,Z 354.854,A -85,B 0,C 180,E1 -549.769,E2 -549.769} C_VEL
LIN {X 0,Y 602.147,Z 347.211,A -85,B 0,C 180,E1 -550.301,E2 -550.301} C_VEL
LIN {X 0,Y 601.521,Z 342.149,A -85,B 0,C 180,E1 -550.594,E2 -550.594} C_VEL
LIN {X 0,Y 601.542,Z 331.57,A -85,B 0,C 180,E1 -551.093,E2 -551.093} C_VEL
LIN {X 0,Y 601.549,Z 319.073,A -85,B 0,C 180,E1 -551.541,E2 -551.541} C_VEL
LIN {X 0,Y 601.566,Z 305.843,A -85,B 0,C 180,E1 -551.861,E2 -551.861} C_VEL
LIN {X 0,Y 601.61,Z 285.255,A -85,B 0,C 180,E1 -552.139,E2 -552.139} C_VEL
LIN {X 0,Y 601.484,Z 195.803,A -85,B 0,C 180,E1 -553.213,E2 -553.213} C_VEL
LIN {X 0,Y 601.442,Z 195.08,A -85,B 0,C 180,E1 -553.257,E2 -553.257} C_VEL
LIN {X 0,Y 601.469,Z 175.352,A -85,B 0,C 180,E1 -555.938,E2 -555.938} C_VEL
LIN {X 0,Y 601.568,Z 155.836,A -85,B 0,C 180,E1 -558.622,E2 -558.622} C_VEL
LIN {X 0,Y 601.636,Z 134.621,A -85,B 0,C 180,E1 -561.59,E2 -561.59} C_VEL
LIN {X 0,Y 601.446,Z 127.477,A -85,B 0,C 180,E1 -562.611,E2 -562.611} C_VEL
LIN {X 0,Y 601.409,Z 127.194,A -85,B 0,C 180,E1 -562.683,E2 -562.683} C_VEL
LIN {X 0,Y 601.392,Z 127.194,A -85,B 0,C 180,E1 -564.879,E2 -564.879} C_VEL
LIN {X 0,Y 601.405,Z 127.199,A -85,B 0,C 180,E1 -567.36,E2 -567.36} C_VEL
LIN {X 0,Y 601.409,Z 127.191,A -85,B 0,C 180,E1 -570.165,E2 -570.165} C_VEL
LIN {X 0,Y 601.407,Z 127.192,A -85,B 0,C 180,E1 -572.712,E2 -572.712} C_VEL
LIN {X 0,Y 601.385,Z 127.2,A -85,B 0,C 180,E1 -575.11,E2 -575.11} C_VEL
LIN {X 0,Y 601.437,Z 127.194,A -85,B 0,C 180,E1 -577.419,E2 -577.419} C_VEL
LIN {X 0,Y 601.407,Z 127.19,A -85,B 0,C 180,E1 -579.996,E2 -579.996} C_VEL
LIN {X 0,Y 601.387,Z 127.196,A -85,B 0,C 180,E1 -582.673,E2 -582.673} C_VEL
LIN {X 0,Y 601.431,Z 127.191,A -85,B 0,C 180,E1 -585.482,E2 -585.482} C_VEL
LIN {X 0,Y 601.419,Z 127.191,A -85,B 0,C 180,E1 -588.408,E2 -588.408} C_VEL
LIN {X 0,Y 601.409,Z 127.2,A -85,B 0,C 180,E1 -590.873,E2 -590.873} C_VEL
LIN {X 0,Y 601.405,Z 127.193,A -85,B 0,C 180,E1 -593.416,E2 -593.416} C_VEL
LIN {X 0,Y 601.42,Z 127.19,A -85,B 0,C 180,E1 -596.066,E2 -596.066} C_VEL
LIN {X 0,Y 601.422,Z 127.196,A -85,B 0,C 180,E1 -598.545,E2 -598.545} C_VEL
LIN {X 0,Y 601.434,Z 127.188,A -85,B 0,C 180,E1 -601.373,E2 -601.373} C_VEL
LIN {X 0,Y 601.401,Z 127.192,A -85,B 0,C 180,E1 -603.635,E2 -603.635} C_VEL
LIN {X 0,Y 601.417,Z 127.199,A -85,B 0,C 180,E1 -606.589,E2 -606.589} C_VEL
LIN {X 0,Y 601.453,Z 127.334,A -85,B 0,C 180,E1 -607.453,E2 -607.453} C_VEL
LIN {X 0,Y 601.676,Z 133.075,A -85,B 0,C 180,E1 -608.23,E2 -608.23} C_VEL
LIN {X 0,Y 601.595,Z 153.316,A -85,B 0,C 180,E1 -610.906,E2 -610.906} C_VEL
LIN {X 0,Y 601.581,Z 156.853,A -85,B 0,C 180,E1 -611.369,E2 -611.369} C_VEL
LIN {X 0,Y 601.985,Z 160.803,A -85,B 0,C 180,E1 -611.442,E2 -611.442} C_VEL
LIN {X 0,Y 601.864,Z 321.669,A -85,B 0,C 180,E1 -613.429,E2 -613.429} C_VEL
LIN {X 0,Y 601.827,Z 337.633,A -85,B 0,C 180,E1 -613.767,E2 -613.767} C_VEL
LIN {X 0,Y 601.754,Z 352.94,A -85,B 0,C 180,E1 -614.243,E2 -614.243} C_VEL
LIN {X 0,Y 601.713,Z 365.719,A -85,B 0,C 180,E1 -614.763,E2 -614.763} C_VEL
LIN {X 0,Y 601.658,Z 379.397,A -85,B 0,C 180,E1 -615.454,E2 -615.454} C_VEL
LIN {X 0,Y 601.617,Z 392.79,A -85,B 0,C 180,E1 -616.283,E2 -616.283} C_VEL
LIN {X 0,Y 601.532,Z 404.722,A -85,B 0,C 180,E1 -617.174,E2 -617.174} C_VEL
LIN {X 0,Y 601.489,Z 416.262,A -85,B 0,C 180,E1 -618.2,E2 -618.2} C_VEL
LIN {X 0,Y 601.43,Z 425.994,A -85,B 0,C 180,E1 -619.223,E2 -619.223} C_VEL
LIN {X 0,Y 601.429,Z 435.526,A -85,B 0,C 180,E1 -620.414,E2 -620.414} C_VEL
LIN {X 0,Y 601.378,Z 443.451,A -85,B 0,C 180,E1 -621.599,E2 -621.599} C_VEL
LIN {X 0,Y 601.369,Z 450.871,A -85,B 0,C 180,E1 -622.951,E2 -622.951} C_VEL
LIN {X 0,Y 601.373,Z 456.76,A -85,B 0,C 180,E1 -624.298,E2 -624.298} C_VEL
LIN {X 0,Y 601.328,Z 460.241,A -85,B 0,C 180,E1 -625.306,E2 -625.306} C_VEL
LIN {X 0,Y 601.336,Z 463.792,A -85,B 0,C 180,E1 -626.649,E2 -626.649} C_VEL
LIN {X 0,Y 601.343,Z 466.136,A -85,B 0,C 180,E1 -627.99,E2 -627.99} C_VEL
LIN {X 0,Y 601.334,Z 467.327,A -85,B 0,C 180,E1 -629.33,E2 -629.33} C_VEL
LIN {X 0,Y 601.336,Z 467.36,A -85,B 0,C 180,E1 -630.669,E2 -630.669} C_VEL
LIN {X 0,Y 601.343,Z 466.243,A -85,B 0,C 180,E1 -632.008,E2 -632.008} C_VEL
LIN {X 0,Y 601.339,Z 463.988,A -85,B 0,C 180,E1 -633.349,E2 -633.349} C_VEL
LIN {X 0,Y 601.328,Z 460.53,A -85,B 0,C 180,E1 -634.692,E2 -634.692} C_VEL
LIN {X 0,Y 601.358,Z 455.796,A -85,B 0,C 180,E1 -636.037,E2 -636.037} C_VEL
LIN {X 0,Y 601.365,Z 449.664,A -85,B 0,C 180,E1 -637.385,E2 -637.385} C_VEL
LIN {X 0,Y 601.389,Z 441.959,A -85,B 0,C 180,E1 -638.737,E2 -638.737} C_VEL
LIN {X 0,Y 601.427,Z 433.717,A -85,B 0,C 180,E1 -639.924,E2 -639.924} C_VEL
LIN {X 0,Y 601.443,Z 424.651,A -85,B 0,C 180,E1 -641.02,E2 -641.02} C_VEL
LIN {X 0,Y 601.514,Z 413.658,A -85,B 0,C 180,E1 -642.139,E2 -642.139} C_VEL
LIN {X 0,Y 601.57,Z 401.611,A -85,B 0,C 180,E1 -643.167,E2 -643.167} C_VEL
LIN {X 0,Y 601.63,Z 388.149,A -85,B 0,C 180,E1 -644.114,E2 -644.114} C_VEL
LIN {X 0,Y 601.677,Z 374.75,A -85,B 0,C 180,E1 -644.89,E2 -644.89} C_VEL
LIN {X 0,Y 601.756,Z 359.853,A -85,B 0,C 180,E1 -645.581,E2 -645.581} C_VEL
LIN {X 0,Y 601.807,Z 345.317,A -85,B 0,C 180,E1 -646.101,E2 -646.101} C_VEL
LIN {X 0,Y 601.85,Z 330.827,A -85,B 0,C 180,E1 -646.484,E2 -646.484} C_VEL
LIN {X 0,Y 601.894,Z 315.977,A -85,B 0,C 180,E1 -646.745,E2 -646.745} C_VEL
LIN {X 0,Y 601.911,Z 158.665,A -85,B 0,C 180,E1 -648.677,E2 -648.677} C_VEL
LIN {X 0,Y 601.576,Z 156.803,A -85,B 0,C 180,E1 -648.727,E2 -648.727} C_VEL
LIN {X 0,Y 601.669,Z 135.113,A -85,B 0,C 180,E1 -651.588,E2 -651.588} C_VEL
LIN {X 0,Y 601.448,Z 127.242,A -85,B 0,C 180,E1 -652.65,E2 -652.65} C_VEL
LIN {X 0,Y 601.4,Z 127.193,A -85,B 0,C 180,E1 -654.877,E2 -654.877} C_VEL
LIN {X 0,Y 601.409,Z 127.198,A -85,B 0,C 180,E1 -657.361,E2 -657.361} C_VEL
LIN {X 0,Y 601.424,Z 127.19,A -85,B 0,C 180,E1 -660.148,E2 -660.148} C_VEL
LIN {X 0,Y 601.425,Z 127.188,A -85,B 0,C 180,E1 -662.716,E2 -662.716} C_VEL
LIN {X 0,Y 601.406,Z 127.195,A -85,B 0,C 180,E1 -665.113,E2 -665.113} C_VEL
LIN {X 0,Y 601.431,Z 127.198,A -85,B 0,C 180,E1 -667.418,E2 -667.418} C_VEL
LIN {X 0,Y 601.405,Z 127.191,A -85,B 0,C 180,E1 -669.994,E2 -669.994} C_VEL
LIN {X 0,Y 601.409,Z 127.191,A -85,B 0,C 180,E1 -672.669,E2 -672.669} C_VEL
LIN {X 0,Y 601.419,Z 127.196,A -85,B 0,C 180,E1 -675.481,E2 -675.481} C_VEL
LIN {X 0,Y 601.418,Z 127.189,A -85,B 0,C 180,E1 -678.406,E2 -678.406} C_VEL
LIN {X 0,Y 601.43,Z 127.192,A -85,B 0,C 180,E1 -680.875,E2 -680.875} C_VEL
LIN {X 0,Y 601.438,Z 127.188,A -85,B 0,C 180,E1 -683.733,E2 -683.733} C_VEL
LIN {X 0,Y 601.426,Z 127.187,A -85,B 0,C 180,E1 -686.063,E2 -686.063} C_VEL
LIN {X 0,Y 601.433,Z 127.189,A -85,B 0,C 180,E1 -688.541,E2 -688.541} C_VEL
LIN {X 0,Y 601.429,Z 127.193,A -85,B 0,C 180,E1 -691.373,E2 -691.373} C_VEL
LIN {X 0,Y 601.398,Z 127.193,A -85,B 0,C 180,E1 -693.636,E2 -693.636} C_VEL
LIN {X 0,Y 601.415,Z 127.192,A -85,B 0,C 180,E1 -696.589,E2 -696.589} C_VEL
LIN {X 0,Y 601.427,Z 127.19,A -85,B 0,C 180,E1 -699.478,E2 -699.478} C_VEL
LIN {X 0,Y 601.392,Z 127.193,A -85,B 0,C 180,E1 -702.311,E2 -702.311} C_VEL
LIN {X 0,Y 601.411,Z 127.192,A -85,B 0,C 180,E1 -704.409,E2 -704.409} C_VEL
LIN {X 0,Y 601.421,Z 127.193,A -85,B 0,C 180,E1 -707.172,E2 -707.172} C_VEL
LIN {X 0,Y 601.424,Z 127.188,A -85,B 0,C 180,E1 -709.905,E2 -709.905} C_VEL
LIN {X 0,Y 601.445,Z 127.192,A -85,B 0,C 180,E1 -712.615,E2 -712.615} C_VEL
LIN {X 0,Y 601.425,Z 127.19,A -85,B 0,C 180,E1 -715.308,E2 -715.308} C_VEL
LIN {X 0,Y 601.411,Z 127.19,A -85,B 0,C 180,E1 -717.991,E2 -717.991} C_VEL
LIN {X 0,Y 601.451,Z 127.194,A -85,B 0,C 180,E1 -720.669,E2 -720.669} C_VEL
LIN {X 0,Y 601.429,Z 127.188,A -85,B 0,C 180,E1 -723.349,E2 -723.349} C_VEL
LIN {X 0,Y 601.398,Z 127.193,A -85,B 0,C 180,E1 -726.037,E2 -726.037} C_VEL
LIN {X 0,Y 601.436,Z 127.194,A -85,B 0,C 180,E1 -728.738,E2 -728.738} C_VEL
LIN {X 0,Y 601.426,Z 127.187,A -85,B 0,C 180,E1 -731.458,E2 -731.458} C_VEL
LIN {X 0,Y 601.409,Z 127.194,A -85,B 0,C 180,E1 -734.206,E2 -734.206} C_VEL
LIN {X 0,Y 601.428,Z 127.19,A -85,B 0,C 180,E1 -736.986,E2 -736.986} C_VEL
LIN {X 0,Y 601.399,Z 127.192,A -85,B 0,C 180,E1 -739.81,E2 -739.81} C_VEL
LIN {X 0,Y 601.446,Z 127.19,A -85,B 0,C 180,E1 -742.682,E2 -742.682} C_VEL
LIN {X 0,Y 601.399,Z 127.193,A -85,B 0,C 180,E1 -744.879,E2 -744.879} C_VEL
LIN {X 0,Y 601.415,Z 127.192,A -85,B 0,C 180,E1 -747.868,E2 -747.868} C_VEL
LIN {X 0,Y 601.418,Z 127.197,A -85,B 0,C 180,E1 -750.165,E2 -750.165} C_VEL
LIN {X 0,Y 601.42,Z 127.191,A -85,B 0,C 180,E1 -752.717,E2 -752.717} C_VEL
LIN {X 0,Y 601.406,Z 127.19,A -85,B 0,C 180,E1 -755.116,E2 -755.116} C_VEL
LIN {X 0,Y 601.426,Z 127.188,A -85,B 0,C 180,E1 -757.42,E2 -757.42} C_VEL
LIN {X 0,Y 601.4,Z 127.198,A -85,B 0,C 180,E1 -759.996,E2 -759.996} C_VEL
LIN {X 0,Y 601.406,Z 127.192,A -85,B 0,C 180,E1 -762.671,E2 -762.671} C_VEL
LIN {X 0,Y 601.418,Z 127.191,A -85,B 0,C 180,E1 -765.483,E2 -765.483} C_VEL
LIN {X 0,Y 601.422,Z 127.193,A -85,B 0,C 180,E1 -768.407,E2 -768.407} C_VEL
LIN {X 0,Y 601.426,Z 127.188,A -85,B 0,C 180,E1 -770.876,E2 -770.876} C_VEL
LIN {X 0,Y 601.435,Z 127.193,A -85,B 0,C 180,E1 -773.735,E2 -773.735} C_VEL
LIN {X 0,Y 601.427,Z 127.188,A -85,B 0,C 180,E1 -776.688,E2 -776.688} C_VEL
LIN {X 0,Y 601.445,Z 127.196,A -85,B 0,C 180,E1 -779.849,E2 -779.849} C_VEL
LIN {X 0,Y 601.441,Z 127.289,A -85,B 0,C 180,E1 -782.199,E2 -782.199} C_VEL
LIN {X 0,Y 602.283,Z 130.212,A -85,B 0,C 180,E1 -782.478,E2 -782.478} C_VEL
LIN {X 0,Y 602.126,Z 162.562,A -85,B 0,C 180,E1 -785.062,E2 -785.062} C_VEL
LIN {X 0,Y 601.966,Z 199.799,A -85,B 0,C 180,E1 -787.974,E2 -787.974} C_VEL
LIN {X 0,Y 601.792,Z 237.016,A -85,B 0,C 180,E1 -790.826,E2 -790.826} C_VEL
LIN {X 0,Y 601.786,Z 243.163,A -85,B 0,C 180,E1 -791.293,E2 -791.293} C_VEL
LIN {X 0,Y 602.01,Z 252.171,A -85,B 0,C 180,E1 -791.414,E2 -791.414} C_VEL
LIN {X 0,Y 601.873,Z 412.584,A -85,B 0,C 180,E1 -793.398,E2 -793.398} C_VEL
LIN {X 0,Y 601.849,Z 427.749,A -85,B 0,C 180,E1 -793.726,E2 -793.726} C_VEL
LIN {X 0,Y 601.778,Z 443.075,A -85,B 0,C 180,E1 -794.202,E2 -794.202} C_VEL
LIN {X 0,Y 601.719,Z 456.783,A -85,B 0,C 180,E1 -794.765,E2 -794.765} C_VEL
LIN {X 0,Y 601.664,Z 470.252,A -85,B 0,C 180,E1 -795.456,E2 -795.456} C_VEL
LIN {X 0,Y 601.617,Z 483.459,A -85,B 0,C 180,E1 -796.284,E2 -796.284} C_VEL
LIN {X 0,Y 601.531,Z 495.297,A -85,B 0,C 180,E1 -797.175,E2 -797.175} C_VEL
LIN {X 0,Y 601.487,Z 506.758,A -85,B 0,C 180,E1 -798.202,E2 -798.202} C_VEL
LIN {X 0,Y 601.431,Z 516.398,A -85,B 0,C 180,E1 -799.225,E2 -799.225} C_VEL
LIN {X 0,Y 601.428,Z 525.862,A -85,B 0,C 180,E1 -800.415,E2 -800.415} C_VEL
LIN {X 0,Y 601.369,Z 533.736,A -85,B 0,C 180,E1 -801.601,E2 -801.601} C_VEL
LIN {X 0,Y 601.368,Z 541.092,A -85,B 0,C 180,E1 -802.952,E2 -802.952} C_VEL
LIN {X 0,Y 601.373,Z 546.927,A -85,B 0,C 180,E1 -804.3,E2 -804.3} C_VEL
LIN {X 0,Y 601.33,Z 550.386,A -85,B 0,C 180,E1 -805.308,E2 -805.308} C_VEL
LIN {X 0,Y 601.337,Z 553.888,A -85,B 0,C 180,E1 -806.651,E2 -806.651} C_VEL
LIN {X 0,Y 601.342,Z 556.193,A -85,B 0,C 180,E1 -807.992,E2 -807.992} C_VEL
LIN {X 0,Y 601.337,Z 557.35,A -85,B 0,C 180,E1 -809.331,E2 -809.331} C_VEL
LIN {X 0,Y 601.337,Z 557.35,A -85,B 0,C 180,E1 -810.67,E2 -810.67} C_VEL
LIN {X 0,Y 601.343,Z 556.191,A -85,B 0,C 180,E1 -812.01,E2 -812.01} C_VEL
LIN {X 0,Y 601.337,Z 553.884,A -85,B 0,C 180,E1 -813.351,E2 -813.351} C_VEL
LIN {X 0,Y 601.33,Z 550.381,A -85,B 0,C 180,E1 -814.694,E2 -814.694} C_VEL
LIN {X 0,Y 601.357,Z 545.604,A -85,B 0,C 180,E1 -816.038,E2 -816.038} C_VEL
LIN {X 0,Y 601.366,Z 539.421,A -85,B 0,C 180,E1 -817.387,E2 -817.387} C_VEL
LIN {X 0,Y 601.389,Z 531.648,A -85,B 0,C 180,E1 -818.739,E2 -818.739} C_VEL
LIN {X 0,Y 601.427,Z 523.364,A -85,B 0,C 180,E1 -819.926,E2 -819.926} C_VEL
LIN {X 0,Y 601.461,Z 512.925,A -85,B 0,C 180,E1 -821.165,E2 -821.165} C_VEL
LIN {X 0,Y 601.514,Z 503.184,A -85,B 0,C 180,E1 -822.141,E2 -822.141} C_VEL
LIN {X 0,Y 601.57,Z 491.006,A -85,B 0,C 180,E1 -823.169,E2 -823.169} C_VEL
LIN {X 0,Y 601.608,Z 479.065,A -85,B 0,C 180,E1 -824.012,E2 -824.012} C_VEL
LIN {X 0,Y 601.676,Z 465.512,A -85,B 0,C 180,E1 -824.805,E2 -824.805} C_VEL
LIN {X 0,Y 601.772,Z 450.824,A -85,B 0,C 180,E1 -825.496,E2 -825.496} C_VEL
LIN {X 0,Y 601.807,Z 436.595,A -85,B 0,C 180,E1 -826.016,E2 -826.016} C_VEL
LIN {X 0,Y 601.85,Z 421.729,A -85,B 0,C 180,E1 -826.419,E2 -826.419} C_VEL
LIN {X 0,Y 601.861,Z 406.881,A -85,B 0,C 180,E1 -826.687,E2 -826.687} C_VEL
LIN {X 0,Y 602.014,Z 245.161,A -85,B 0,C 180,E1 -828.672,E2 -828.672} C_VEL
LIN {X 0,Y 601.761,Z 242.964,A -85,B 0,C 180,E1 -828.723,E2 -828.723} C_VEL
LIN {X 0,Y 601.931,Z 207.908,A -85,B 0,C 180,E1 -831.4,E2 -831.4} C_VEL
LIN {X 0,Y 602.078,Z 173.008,A -85,B 0,C 180,E1 -834.115,E2 -834.115} C_VEL
LIN {X 0,Y 602.237,Z 140.434,A -85,B 0,C 180,E1 -836.699,E2 -836.699} C_VEL
LIN {X 0,Y 602.145,Z 129.662,A -85,B 0,C 180,E1 -837.573,E2 -837.573} C_VEL
LIN {X 0,Y 601.429,Z 127.197,A -85,B 0,C 180,E1 -837.835,E2 -837.835} C_VEL
LIN {X 0,Y 601.408,Z 127.199,A -85,B 0,C 180,E1 -840.166,E2 -840.166} C_VEL
LIN {X 0,Y 601.4,Z 127.193,A -85,B 0,C 180,E1 -842.712,E2 -842.712} C_VEL
LIN {X 0,Y 601.38,Z 127.196,A -85,B 0,C 180,E1 -845.11,E2 -845.11} C_VEL
LIN {X 0,Y 601.431,Z 127.193,A -85,B 0,C 180,E1 -847.42,E2 -847.42} C_VEL
LIN {X 0,Y 601.379,Z 127.198,A -85,B 0,C 180,E1 -849.998,E2 -849.998} C_VEL
LIN {X 0,Y 601.359,Z 127.197,A -85,B 0,C 180,E1 -852.585,E2 -852.585} C_VEL
LIN {X 0,Y 601.366,Z 127.196,A -85,B 0,C 180,E1 -854.53,E2 -854.53} C_VEL
LIN {X 0,Y 601.37,Z 127.205,A -85,B 0,C 180,E1 -857.326,E2 -857.326} C_VEL
LIN {X 0,Y 601.372,Z 127.196,A -85,B 0,C 180,E1 -860.002,E2 -860.002} C_VEL
LIN {X 0,Y 601.396,Z 127.196,A -85,B 0,C 180,E1 -862.624,E2 -862.624} C_VEL
LIN {X 0,Y 601.403,Z 127.192,A -85,B 0,C 180,E1 -865.88,E2 -865.88} C_VEL
LIN {X 0,Y 601.394,Z 127.198,A -85,B 0,C 180,E1 -868.55,E2 -868.55} C_VEL
LIN {X 0,Y 601.402,Z 127.193,A -85,B 0,C 180,E1 -871.372,E2 -871.372} C_VEL
LIN {X 0,Y 601.384,Z 127.195,A -85,B 0,C 180,E1 -873.635,E2 -873.635} C_VEL
LIN {X 0,Y 601.404,Z 127.194,A -85,B 0,C 180,E1 -875.857,E2 -875.857} C_VEL
LIN {X 0,Y 601.387,Z 127.206,A -85,B 0,C 180,E1 -877.438,E2 -877.438} C_VEL
LIN {X 0,Y 601.656,Z 135.257,A -85,B 0,C 180,E1 -878.59,E2 -878.59} C_VEL
LIN {X 0,Y 601.553,Z 153.513,A -85,B 0,C 180,E1 -881.144,E2 -881.144} C_VEL
LIN {X 0,Y 601.513,Z 173.423,A -85,B 0,C 180,E1 -883.89,E2 -883.89} C_VEL
LIN {X 0,Y 601.456,Z 195.479,A -85,B 0,C 180,E1 -886.872,E2 -886.872} C_VEL
LIN {X 0,Y 601.654,Z 270.589,A -85,B 0,C 180,E1 -887.777,E2 -887.777} C_VEL
LIN {X 0,Y 601.608,Z 304.471,A -85,B 0,C 180,E1 -888.204,E2 -888.204} C_VEL
LIN {X 0,Y 601.592,Z 318.159,A -85,B 0,C 180,E1 -888.524,E2 -888.524} C_VEL
LIN {X 0,Y 601.536,Z 330.122,A -85,B 0,C 180,E1 -888.936,E2 -888.936} C_VEL
LIN {X 0,Y 601.497,Z 341.879,A -85,B 0,C 180,E1 -889.481,E2 -889.481} C_VEL
LIN {X 0,Y 601.446,Z 353.302,A -85,B 0,C 180,E1 -890.16,E2 -890.16} C_VEL
LIN {X 0,Y 601.438,Z 363.594,A -85,B 0,C 180,E1 -890.924,E2 -890.924} C_VEL
LIN {X 0,Y 601.411,Z 372.855,A -85,B 0,C 180,E1 -891.77,E2 -891.77} C_VEL
LIN {X 0,Y 601.389,Z 381.829,A -85,B 0,C 180,E1 -892.783,E2 -892.783} C_VEL
LIN {X 0,Y 601.376,Z 388.968,A -85,B 0,C 180,E1 -893.781,E2 -893.781} C_VEL
LIN {X 0,Y 601.372,Z 393.938,A -85,B 0,C 180,E1 -894.635,E2 -894.635} C_VEL
LIN {X 0,Y 601.355,Z 398.681,A -85,B 0,C 180,E1 -895.643,E2 -895.643} C_VEL
LIN {X 0,Y 601.345,Z 402.315,A -85,B 0,C 180,E1 -896.65,E2 -896.65} C_VEL
LIN {X 0,Y 601.324,Z 404.193,A -85,B 0,C 180,E1 -897.321,E2 -897.321} C_VEL
LIN {X 0,Y 601.341,Z 405.627,A -85,B 0,C 180,E1 -897.991,E2 -897.991} C_VEL
LIN {X 0,Y 601.34,Z 407.253,A -85,B 0,C 180,E1 -899.33,E2 -899.33} C_VEL
LIN {X 0,Y 601.335,Z 407.496,A -85,B 0,C 180,E1 -900,E2 -900} C_VEL
LIN {X 0,Y 601.339,Z 407.315,A -85,B 0,C 180,E1 -900.67,E2 -900.67} C_VEL
LIN {X 0,Y 601.34,Z 405.776,A -85,B 0,C 180,E1 -902.009,E2 -902.009} C_VEL
LIN {X 0,Y 601.326,Z 404.417,A -85,B 0,C 180,E1 -902.68,E2 -902.68} C_VEL
LIN {X 0,Y 601.368,Z 401.539,A -85,B 0,C 180,E1 -903.685,E2 -903.685} C_VEL
LIN {X 0,Y 601.337,Z 397.64,A -85,B 0,C 180,E1 -904.693,E2 -904.693} C_VEL
LIN {X 0,Y 601.373,Z 392.61,A -85,B 0,C 180,E1 -905.701,E2 -905.701} C_VEL
LIN {X 0,Y 601.383,Z 386.291,A -85,B 0,C 180,E1 -906.711,E2 -906.711} C_VEL
LIN {X 0,Y 601.396,Z 378.374,A -85,B 0,C 180,E1 -907.723,E2 -907.723} C_VEL
LIN {X 0,Y 601.437,Z 368.529,A -85,B 0,C 180,E1 -908.738,E2 -908.738} C_VEL
LIN {X 0,Y 601.446,Z 358.206,A -85,B 0,C 180,E1 -909.585,E2 -909.585} C_VEL
LIN {X 0,Y 601.494,Z 346.587,A -85,B 0,C 180,E1 -910.349,E2 -910.349} C_VEL
LIN {X 0,Y 601.521,Z 342.149,A -85,B 0,C 180,E1 -910.594,E2 -910.594} C_VEL
LIN {X 0,Y 600.895,Z 337.02,A -85,B 0,C 180,E1 -910.868,E2 -910.868} C_VEL
LIN {X 0,Y 598.086,Z 328.573,A -85,B 0,C 180,E1 -911.288,E2 -911.288} C_VEL
LIN {X 0,Y 595.262,Z 319.831,A -85,B 0,C 180,E1 -911.644,E2 -911.644} C_VEL
LIN {X 0,Y 594.607,Z 314.244,A -85,B 0,C 180,E1 -911.814,E2 -911.814} C_VEL
LIN {X 0,Y 594.664,Z 302.226,A -85,B 0,C 180,E1 -912.066,E2 -912.066} C_VEL
LIN {X 0,Y 594.622,Z 196.877,A -85,B 0,C 180,E1 -913.355,E2 -913.355} C_VEL
LIN {X 0,Y 594.401,Z 195.235,A -85,B 0,C 180,E1 -913.395,E2 -913.395} C_VEL
LIN {X 0,Y 594.481,Z 176.62,A -85,B 0,C 180,E1 -915.954,E2 -915.954} C_VEL
LIN {X 0,Y 594.584,Z 157.528,A -85,B 0,C 180,E1 -918.611,E2 -918.611} C_VEL
LIN {X 0,Y 594.677,Z 138.354,A -85,B 0,C 180,E1 -921.321,E2 -921.321} C_VEL
LIN {X 0,Y 594.731,Z 130.272,A -85,B 0,C 180,E1 -922.48,E2 -922.48} C_VEL
LIN {X 0,Y 594.362,Z 128.073,A -85,B 0,C 180,E1 -922.851,E2 -922.851} C_VEL
LIN {X 0,Y 594.373,Z 128.072,A -85,B 0,C 180,E1 -925.193,E2 -925.193} C_VEL
LIN {X 0,Y 594.353,Z 128.08,A -85,B 0,C 180,E1 -927.52,E2 -927.52} C_VEL
LIN {X 0,Y 594.373,Z 128.067,A -85,B 0,C 180,E1 -930.325,E2 -930.325} C_VEL
LIN {X 0,Y 594.379,Z 128.07,A -85,B 0,C 180,E1 -932.95,E2 -932.95} C_VEL
LIN {X 0,Y 594.35,Z 128.078,A -85,B 0,C 180,E1 -935.409,E2 -935.409} C_VEL
LIN {X 0,Y 594.382,Z 128.067,A -85,B 0,C 180,E1 -937.941,E2 -937.941} C_VEL
LIN {X 0,Y 594.373,Z 128.07,A -85,B 0,C 180,E1 -940.821,E2 -940.821} C_VEL
LIN {X 0,Y 594.365,Z 128.068,A -85,B 0,C 180,E1 -943.838,E2 -943.838} C_VEL
LIN {X 0,Y 594.357,Z 128.074,A -85,B 0,C 180,E1 -946.699,E2 -946.699} C_VEL
LIN {X 0,Y 594.369,Z 128.07,A -85,B 0,C 180,E1 -949.432,E2 -949.432} C_VEL
LIN {X 0,Y 594.391,Z 128.067,A -85,B 0,C 180,E1 -952.392,E2 -952.392} C_VEL
LIN {X 0,Y 594.379,Z 128.068,A -85,B 0,C 180,E1 -955.419,E2 -955.419} C_VEL
LIN {X 0,Y 594.379,Z 128.071,A -85,B 0,C 180,E1 -958.357,E2 -958.357} C_VEL
LIN {X 0,Y 594.387,Z 128.069,A -85,B 0,C 180,E1 -961.042,E2 -961.042} C_VEL
LIN {X 0,Y 594.384,Z 128.068,A -85,B 0,C 180,E1 -963.978,E2 -963.978} C_VEL
LIN {X 0,Y 594.386,Z 128.073,A -85,B 0,C 180,E1 -966.295,E2 -966.295} C_VEL
LIN {X 0,Y 594.375,Z 128.114,A -85,B 0,C 180,E1 -967.275,E2 -967.275} C_VEL
LIN {X 0,Y 594.756,Z 133.08,A -85,B 0,C 180,E1 -967.964,E2 -967.964} C_VEL
LIN {X 0,Y 594.655,Z 153.321,A -85,B 0,C 180,E1 -970.675,E2 -970.675} C_VEL
LIN {X 0,Y 594.62,Z 156.919,A -85,B 0,C 180,E1 -971.151,E2 -971.151} C_VEL
LIN {X 0,Y 595.272,Z 161.037,A -85,B 0,C 180,E1 -971.227,E2 -971.227} C_VEL
LIN {X 0,Y 595.081,Z 322.037,A -85,B 0,C 180,E1 -973.241,E2 -973.241} C_VEL
LIN {X 0,Y 595.022,Z 337.655,A -85,B 0,C 180,E1 -973.576,E2 -973.576} C_VEL
LIN {X 0,Y 594.912,Z 352.928,A -85,B 0,C 180,E1 -974.057,E2 -974.057} C_VEL
LIN {X 0,Y 594.832,Z 365.713,A -85,B 0,C 180,E1 -974.582,E2 -974.582} C_VEL
LIN {X 0,Y 594.732,Z 379.406,A -85,B 0,C 180,E1 -975.281,E2 -975.281} C_VEL
LIN {X 0,Y 594.683,Z 392.14,A -85,B 0,C 180,E1 -976.074,E2 -976.074} C_VEL
LIN {X 0,Y 594.56,Z 404.731,A -85,B 0,C 180,E1 -977.021,E2 -977.021} C_VEL
LIN {X 0,Y 594.466,Z 416.261,A -85,B 0,C 180,E1 -978.059,E2 -978.059} C_VEL
LIN {X 0,Y 594.39,Z 426.002,A -85,B 0,C 180,E1 -979.094,E2 -979.094} C_VEL
LIN {X 0,Y 594.382,Z 435.535,A -85,B 0,C 180,E1 -980.299,E2 -980.299} C_VEL
LIN {X 0,Y 594.318,Z 443.451,A -85,B 0,C 180,E1 -981.499,E2 -981.499} C_VEL
LIN {X 0,Y 594.293,Z 450.875,A -85,B 0,C 180,E1 -982.866,E2 -982.866} C_VEL
LIN {X 0,Y 594.299,Z 456.766,A -85,B 0,C 180,E1 -984.23,E2 -984.23} C_VEL
LIN {X 0,Y 594.23,Z 460.245,A -85,B 0,C 180,E1 -985.25,E2 -985.25} C_VEL
LIN {X 0,Y 594.256,Z 463.797,A -85,B 0,C 180,E1 -986.609,E2 -986.609} C_VEL
LIN {X 0,Y 594.241,Z 466.135,A -85,B 0,C 180,E1 -987.966,E2 -987.966} C_VEL
LIN {X 0,Y 594.235,Z 467.32,A -85,B 0,C 180,E1 -989.321,E2 -989.321} C_VEL
LIN {X 0,Y 594.236,Z 467.353,A -85,B 0,C 180,E1 -990.677,E2 -990.677} C_VEL
LIN {X 0,Y 594.242,Z 466.24,A -85,B 0,C 180,E1 -992.032,E2 -992.032} C_VEL
LIN {X 0,Y 594.258,Z 463.991,A -85,B 0,C 180,E1 -993.389,E2 -993.389} C_VEL
LIN {X 0,Y 594.231,Z 460.53,A -85,B 0,C 180,E1 -994.748,E2 -994.748} C_VEL
LIN {X 0,Y 594.279,Z 455.786,A -85,B 0,C 180,E1 -996.109,E2 -996.109} C_VEL
LIN {X 0,Y 594.287,Z 449.652,A -85,B 0,C 180,E1 -997.474,E2 -997.474} C_VEL
LIN {X 0,Y 594.332,Z 441.957,A -85,B 0,C 180,E1 -998.842,E2 -998.842} C_VEL
LIN {X 0,Y 594.387,Z 433.712,A -85,B 0,C 180,E1 -1000.043,E2 -1000.043} C_VEL
LIN {X 0,Y 594.409,Z 423.959,A -85,B 0,C 180,E1 -1001.228,E2 -1001.228} C_VEL
LIN {X 0,Y 594.514,Z 413.643,A -85,B 0,C 180,E1 -1002.285,E2 -1002.285} C_VEL
LIN {X 0,Y 594.579,Z 401.605,A -85,B 0,C 180,E1 -1003.325,E2 -1003.325} C_VEL
LIN {X 0,Y 594.692,Z 388.033,A -85,B 0,C 180,E1 -1004.288,E2 -1004.288} C_VEL
LIN {X 0,Y 594.789,Z 374.721,A -85,B 0,C 180,E1 -1005.066,E2 -1005.066} C_VEL
LIN {X 0,Y 594.88,Z 359.837,A -85,B 0,C 180,E1 -1005.766,E2 -1005.766} C_VEL
LIN {X 0,Y 594.958,Z 345.265,A -85,B 0,C 180,E1 -1006.292,E2 -1006.292} C_VEL
LIN {X 0,Y 595.039,Z 330.569,A -85,B 0,C 180,E1 -1006.683,E2 -1006.683} C_VEL
LIN {X 0,Y 595.109,Z 314.743,A -85,B 0,C 180,E1 -1006.959,E2 -1006.959} C_VEL
LIN {X 0,Y 595.234,Z 159.945,A -85,B 0,C 180,E1 -1008.878,E2 -1008.878} C_VEL
LIN {X 0,Y 594.637,Z 156.895,A -85,B 0,C 180,E1 -1008.942,E2 -1008.942} C_VEL
LIN {X 0,Y 594.764,Z 136.459,A -85,B 0,C 180,E1 -1011.669,E2 -1011.669} C_VEL
LIN {X 0,Y 594.753,Z 130.266,A -85,B 0,C 180,E1 -1012.507,E2 -1012.507} C_VEL
LIN {X 0,Y 594.374,Z 128.072,A -85,B 0,C 180,E1 -1012.852,E2 -1012.852} C_VEL
LIN {X 0,Y 594.376,Z 128.072,A -85,B 0,C 180,E1 -1015.192,E2 -1015.192} C_VEL
LIN {X 0,Y 594.383,Z 128.076,A -85,B 0,C 180,E1 -1017.526,E2 -1017.526} C_VEL
LIN {X 0,Y 594.384,Z 128.066,A -85,B 0,C 180,E1 -1020.327,E2 -1020.327} C_VEL
LIN {X 0,Y 594.377,Z 128.068,A -85,B 0,C 180,E1 -1022.949,E2 -1022.949} C_VEL
LIN {X 0,Y 594.377,Z 128.076,A -85,B 0,C 180,E1 -1025.406,E2 -1025.406} C_VEL
LIN {X 0,Y 594.382,Z 128.068,A -85,B 0,C 180,E1 -1027.94,E2 -1027.94} C_VEL
LIN {X 0,Y 594.375,Z 128.067,A -85,B 0,C 180,E1 -1030.822,E2 -1030.822} C_VEL
LIN {X 0,Y 594.376,Z 128.068,A -85,B 0,C 180,E1 -1033.84,E2 -1033.84} C_VEL
LIN {X 0,Y 594.359,Z 128.07,A -85,B 0,C 180,E1 -1036.7,E2 -1036.7} C_VEL
LIN {X 0,Y 594.366,Z 128.074,A -85,B 0,C 180,E1 -1039.433,E2 -1039.433} C_VEL
LIN {X 0,Y 594.383,Z 128.065,A -85,B 0,C 180,E1 -1042.39,E2 -1042.39} C_VEL
LIN {X 0,Y 594.379,Z 128.068,A -85,B 0,C 180,E1 -1044.67,E2 -1044.67} C_VEL
LIN {X 0,Y 594.37,Z 128.076,A -85,B 0,C 180,E1 -1047.087,E2 -1047.087} C_VEL
LIN {X 0,Y 594.393,Z 128.065,A -85,B 0,C 180,E1 -1049.668,E2 -1049.668} C_VEL
LIN {X 0,Y 594.364,Z 128.07,A -85,B 0,C 180,E1 -1052.538,E2 -1052.538} C_VEL
LIN {X 0,Y 594.37,Z 128.073,A -85,B 0,C 180,E1 -1054.807,E2 -1054.807} C_VEL
LIN {X 0,Y 594.356,Z 128.074,A -85,B 0,C 180,E1 -1057.263,E2 -1057.263} C_VEL
LIN {X 0,Y 594.371,Z 128.066,A -85,B 0,C 180,E1 -1059.946,E2 -1059.946} C_VEL
LIN {X 0,Y 594.382,Z 128.073,A -85,B 0,C 180,E1 -1062.806,E2 -1062.806} C_VEL
LIN {X 0,Y 594.378,Z 128.065,A -85,B 0,C 180,E1 -1065.825,E2 -1065.825} C_VEL
LIN {X 0,Y 594.387,Z 128.067,A -85,B 0,C 180,E1 -1068.404,E2 -1068.404} C_VEL
LIN {X 0,Y 594.395,Z 128.068,A -85,B 0,C 180,E1 -1071.158,E2 -1071.158} C_VEL
LIN {X 0,Y 594.356,Z 128.067,A -85,B 0,C 180,E1 -1073.891,E2 -1073.891} C_VEL
LIN {X 0,Y 594.379,Z 128.074,A -85,B 0,C 180,E1 -1076.611,E2 -1076.611} C_VEL
LIN {X 0,Y 594.419,Z 128.061,A -85,B 0,C 180,E1 -1079.322,E2 -1079.322} C_VEL
LIN {X 0,Y 594.381,Z 128.066,A -85,B 0,C 180,E1 -1082.033,E2 -1082.033} C_VEL
LIN {X 0,Y 594.397,Z 128.071,A -85,B 0,C 180,E1 -1084.748,E2 -1084.748} C_VEL
LIN {X 0,Y 594.393,Z 128.063,A -85,B 0,C 180,E1 -1087.473,E2 -1087.473} C_VEL
LIN {X 0,Y 594.383,Z 128.07,A -85,B 0,C 180,E1 -1090.216,E2 -1090.216} C_VEL
LIN {X 0,Y 594.369,Z 128.069,A -85,B 0,C 180,E1 -1092.983,E2 -1092.983} C_VEL
LIN {X 0,Y 594.361,Z 128.068,A -85,B 0,C 180,E1 -1095.781,E2 -1095.781} C_VEL
LIN {X 0,Y 594.38,Z 128.072,A -85,B 0,C 180,E1 -1098.618,E2 -1098.618} C_VEL
LIN {X 0,Y 594.357,Z 128.068,A -85,B 0,C 180,E1 -1101.504,E2 -1101.504} C_VEL
LIN {X 0,Y 594.378,Z 128.066,A -85,B 0,C 180,E1 -1103.704,E2 -1103.704} C_VEL
LIN {X 0,Y 594.384,Z 128.069,A -85,B 0,C 180,E1 -1106.7,E2 -1106.7} C_VEL
LIN {X 0,Y 594.374,Z 128.066,A -85,B 0,C 180,E1 -1108.999,E2 -1108.999} C_VEL
LIN {X 0,Y 594.383,Z 128.067,A -85,B 0,C 180,E1 -1111.646,E2 -1111.646} C_VEL
LIN {X 0,Y 594.39,Z 128.069,A -85,B 0,C 180,E1 -1114.579,E2 -1114.579} C_VEL
LIN {X 0,Y 594.378,Z 128.066,A -85,B 0,C 180,E1 -1117.087,E2 -1117.087} C_VEL
LIN {X 0,Y 594.353,Z 128.072,A -85,B 0,C 180,E1 -1119.774,E2 -1119.774} C_VEL
LIN {X 0,Y 594.365,Z 128.073,A -85,B 0,C 180,E1 -1122.376,E2 -1122.376} C_VEL
LIN {X 0,Y 594.355,Z 128.069,A -85,B 0,C 180,E1 -1125.192,E2 -1125.192} C_VEL
LIN {X 0,Y 594.359,Z 128.072,A -85,B 0,C 180,E1 -1127.625,E2 -1127.625} C_VEL
LIN {X 0,Y 594.385,Z 128.07,A -85,B 0,C 180,E1 -1130.322,E2 -1130.322} C_VEL
LIN {X 0,Y 594.377,Z 128.066,A -85,B 0,C 180,E1 -1132.914,E2 -1132.914} C_VEL
LIN {X 0,Y 594.377,Z 128.075,A -85,B 0,C 180,E1 -1135.862,E2 -1135.862} C_VEL
LIN {X 0,Y 594.364,Z 128.069,A -85,B 0,C 180,E1 -1138.651,E2 -1138.651} C_VEL
LIN {X 0,Y 594.376,Z 128.068,A -85,B 0,C 180,E1 -1141.043,E2 -1141.043} C_VEL
LIN {X 0,Y 594.391,Z 128.075,A -85,B 0,C 180,E1 -1141.921,E2 -1141.921} C_VEL
LIN {X 0,Y 595.658,Z 132.763,A -85,B 0,C 180,E1 -1142.36,E2 -1142.36} C_VEL
LIN {X 0,Y 595.456,Z 163.725,A -85,B 0,C 180,E1 -1144.857,E2 -1144.857} C_VEL
LIN {X 0,Y 595.2,Z 200.952,A -85,B 0,C 180,E1 -1147.801,E2 -1147.801} C_VEL
LIN {X 0,Y 594.956,Z 238.179,A -85,B 0,C 180,E1 -1150.687,E2 -1150.687} C_VEL
LIN {X 0,Y 594.915,Z 243.11,A -85,B 0,C 180,E1 -1151.065,E2 -1151.065} C_VEL
LIN {X 0,Y 595.318,Z 248.439,A -85,B 0,C 180,E1 -1151.151,E2 -1151.151} C_VEL
LIN {X 0,Y 595.091,Z 412.192,A -85,B 0,C 180,E1 -1153.196,E2 -1153.196} C_VEL
LIN {X 0,Y 595.025,Z 427.748,A -85,B 0,C 180,E1 -1153.534,E2 -1153.534} C_VEL
LIN {X 0,Y 594.951,Z 443.073,A -85,B 0,C 180,E1 -1154.016,E2 -1154.016} C_VEL
LIN {X 0,Y 594.856,Z 456.786,A -85,B 0,C 180,E1 -1154.585,E2 -1154.585} C_VEL
LIN {X 0,Y 594.74,Z 470.255,A -85,B 0,C 180,E1 -1155.283,E2 -1155.283} C_VEL
LIN {X 0,Y 594.679,Z 482.807,A -85,B 0,C 180,E1 -1156.076,E2 -1156.076} C_VEL
LIN {X 0,Y 594.559,Z 495.298,A -85,B 0,C 180,E1 -1157.022,E2 -1157.022} C_VEL
LIN {X 0,Y 594.464,Z 506.758,A -85,B 0,C 180,E1 -1158.061,E2 -1158.061} C_VEL
LIN {X 0,Y 594.388,Z 516.398,A -85,B 0,C 180,E1 -1159.096,E2 -1159.096} C_VEL
LIN {X 0,Y 594.366,Z 525.863,A -85,B 0,C 180,E1 -1160.301,E2 -1160.301} C_VEL
LIN {X 0,Y 594.312,Z 533.737,A -85,B 0,C 180,E1 -1161.5,E2 -1161.5} C_VEL
LIN {X 0,Y 594.291,Z 541.093,A -85,B 0,C 180,E1 -1162.868,E2 -1162.868} C_VEL
LIN {X 0,Y 594.299,Z 546.927,A -85,B 0,C 180,E1 -1164.232,E2 -1164.232} C_VEL
LIN {X 0,Y 594.232,Z 550.386,A -85,B 0,C 180,E1 -1165.252,E2 -1165.252} C_VEL
LIN {X 0,Y 594.256,Z 553.889,A -85,B 0,C 180,E1 -1166.611,E2 -1166.611} C_VEL
LIN {X 0,Y 594.241,Z 556.194,A -85,B 0,C 180,E1 -1167.968,E2 -1167.968} C_VEL
LIN {X 0,Y 594.237,Z 557.35,A -85,B 0,C 180,E1 -1169.323,E2 -1169.323} C_VEL
LIN {X 0,Y 594.237,Z 557.35,A -85,B 0,C 180,E1 -1170.679,E2 -1170.679} C_VEL
LIN {X 0,Y 594.241,Z 556.191,A -85,B 0,C 180,E1 -1172.034,E2 -1172.034} C_VEL
LIN {X 0,Y 594.256,Z 553.884,A -85,B 0,C 180,E1 -1173.391,E2 -1173.391} C_VEL
LIN {X 0,Y 594.232,Z 550.381,A -85,B 0,C 180,E1 -1174.75,E2 -1174.75} C_VEL
LIN {X 0,Y 594.279,Z 545.605,A -85,B 0,C 180,E1 -1176.111,E2 -1176.111} C_VEL
LIN {X 0,Y 594.287,Z 539.42,A -85,B 0,C 180,E1 -1177.475,E2 -1177.475} C_VEL
LIN {X 0,Y 594.331,Z 531.646,A -85,B 0,C 180,E1 -1178.844,E2 -1178.844} C_VEL
LIN {X 0,Y 594.387,Z 523.364,A -85,B 0,C 180,E1 -1180.045,E2 -1180.045} C_VEL
LIN {X 0,Y 594.435,Z 513.552,A -85,B 0,C 180,E1 -1181.232,E2 -1181.232} C_VEL
LIN {X 0,Y 594.531,Z 503.183,A -85,B 0,C 180,E1 -1182.286,E2 -1182.286} C_VEL
LIN {X 0,Y 594.582,Z 491.007,A -85,B 0,C 180,E1 -1183.327,E2 -1183.327} C_VEL
LIN {X 0,Y 594.696,Z 479.062,A -85,B 0,C 180,E1 -1184.178,E2 -1184.178} C_VEL
LIN {X 0,Y 594.777,Z 465.509,A -85,B 0,C 180,E1 -1184.981,E2 -1184.981} C_VEL
LIN {X 0,Y 594.914,Z 450.821,A -85,B 0,C 180,E1 -1185.679,E2 -1185.679} C_VEL
LIN {X 0,Y 594.99,Z 436.595,A -85,B 0,C 180,E1 -1186.205,E2 -1186.205} C_VEL
LIN {X 0,Y 595.047,Z 422.169,A -85,B 0,C 180,E1 -1186.602,E2 -1186.602} C_VEL
LIN {X 0,Y 595.061,Z 406.881,A -85,B 0,C 180,E1 -1186.884,E2 -1186.884} C_VEL
LIN {X 0,Y 595.234,Z 245.453,A -85,B 0,C 180,E1 -1188.889,E2 -1188.889} C_VEL
LIN {X 0,Y 594.922,Z 243.083,A -85,B 0,C 180,E1 -1188.937,E2 -1188.937} C_VEL
LIN {X 0,Y 595.15,Z 209.072,A -85,B 0,C 180,E1 -1191.565,E2 -1191.565} C_VEL
LIN {X 0,Y 595.374,Z 173.008,A -85,B 0,C 180,E1 -1194.404,E2 -1194.404} C_VEL
LIN {X 0,Y 595.621,Z 140.434,A -85,B 0,C 180,E1 -1197.019,E2 -1197.019} C_VEL
LIN {X 0,Y 595.467,Z 131.783,A -85,B 0,C 180,E1 -1197.726,E2 -1197.726} C_VEL
LIN {X 0,Y 594.392,Z 128.075,A -85,B 0,C 180,E1 -1198.08,E2 -1198.08} C_VEL
LIN {X 0,Y 594.368,Z 128.071,A -85,B 0,C 180,E1 -1200.561,E2 -1200.561} C_VEL
LIN {X 0,Y 594.376,Z 128.068,A -85,B 0,C 180,E1 -1202.951,E2 -1202.951} C_VEL
LIN {X 0,Y 594.328,Z 128.077,A -85,B 0,C 180,E1 -1205.411,E2 -1205.411} C_VEL
LIN {X 0,Y 594.357,Z 128.075,A -85,B 0,C 180,E1 -1207.944,E2 -1207.944} C_VEL
LIN {X 0,Y 594.359,Z 128.07,A -85,B 0,C 180,E1 -1210.82,E2 -1210.82} C_VEL
LIN {X 0,Y 594.336,Z 128.076,A -85,B 0,C 180,E1 -1213.836,E2 -1213.836} C_VEL
LIN {X 0,Y 594.34,Z 128.073,A -85,B 0,C 180,E1 -1216.698,E2 -1216.698} C_VEL
LIN {X 0,Y 594.311,Z 128.081,A -85,B 0,C 180,E1 -1219.428,E2 -1219.428} C_VEL
LIN {X 0,Y 594.304,Z 128.076,A -85,B 0,C 180,E1 -1222.053,E2 -1222.053} C_VEL
LIN {X 0,Y 594.316,Z 128.08,A -85,B 0,C 180,E1 -1224.682,E2 -1224.682} C_VEL
LIN {X 0,Y 594.342,Z 128.078,A -85,B 0,C 180,E1 -1227.095,E2 -1227.095} C_VEL
LIN {X 0,Y 594.349,Z 128.071,A -85,B 0,C 180,E1 -1229.679,E2 -1229.679} C_VEL
LIN {X 0,Y 594.325,Z 128.074,A -85,B 0,C 180,E1 -1231.77,E2 -1231.77} C_VEL
LIN {X 0,Y 594.359,Z 128.073,A -85,B 0,C 180,E1 -1234.055,E2 -1234.055} C_VEL
LIN {X 0,Y 594.352,Z 128.077,A -85,B 0,C 180,E1 -1237.032,E2 -1237.032} C_VEL
LIN {X 0,Y 594.37,Z 128.105,A -85,B 0,C 180,E1 -1237.265,E2 -1237.265} C_VEL
LIN {X 0,Y 594.712,Z 133.99,A -85,B 0,C 180,E1 -1238.146,E2 -1238.146} C_VEL
LIN {X 0,Y 594.629,Z 153.411,A -85,B 0,C 180,E1 -1240.902,E2 -1240.902} C_VEL
LIN {X 0,Y 594.512,Z 173.427,A -85,B 0,C 180,E1 -1243.695,E2 -1243.695} C_VEL
LIN {X 0,Y 594.445,Z 195.214,A -85,B 0,C 180,E1 -1246.693,E2 -1246.693} C_VEL
LIN {X 0,Y 594.737,Z 199.099,A -85,B 0,C 180,E1 -1246.765,E2 -1246.765} C_VEL
LIN {X 0,Y 594.678,Z 303.358,A -85,B 0,C 180,E1 -1248.043,E2 -1248.043} C_VEL
LIN {X 0,Y 594.633,Z 316.661,A -85,B 0,C 180,E1 -1248.344,E2 -1248.344} C_VEL
LIN {X 0,Y 594.581,Z 329.908,A -85,B 0,C 180,E1 -1248.796,E2 -1248.796} C_VEL
LIN {X 0,Y 594.515,Z 341.887,A -85,B 0,C 180,E1 -1249.356,E2 -1249.356} C_VEL
LIN {X 0,Y 594.447,Z 353.312,A -85,B 0,C 180,E1 -1250.043,E2 -1250.043} C_VEL
LIN {X 0,Y 594.406,Z 363.602,A -85,B 0,C 180,E1 -1250.815,E2 -1250.815} C_VEL
LIN {X 0,Y 594.373,Z 372.86,A -85,B 0,C 180,E1 -1251.672,E2 -1251.672} C_VEL
LIN {X 0,Y 594.317,Z 381.834,A -85,B 0,C 180,E1 -1252.697,E2 -1252.697} C_VEL
LIN {X 0,Y 594.285,Z 388.356,A -85,B 0,C 180,E1 -1253.612,E2 -1253.612} C_VEL
LIN {X 0,Y 594.289,Z 393.94,A -85,B 0,C 180,E1 -1254.571,E2 -1254.571} C_VEL
LIN {X 0,Y 594.271,Z 398.684,A -85,B 0,C 180,E1 -1255.591,E2 -1255.591} C_VEL
LIN {X 0,Y 594.268,Z 402.317,A -85,B 0,C 180,E1 -1256.61,E2 -1256.61} C_VEL
LIN {X 0,Y 594.225,Z 404.195,A -85,B 0,C 180,E1 -1257.288,E2 -1257.288} C_VEL
LIN {X 0,Y 594.24,Z 405.626,A -85,B 0,C 180,E1 -1257.967,E2 -1257.967} C_VEL
LIN {X 0,Y 594.241,Z 407.253,A -85,B 0,C 180,E1 -1259.322,E2 -1259.322} C_VEL
LIN {X 0,Y 594.236,Z 407.496,A -85,B 0,C 180,E1 -1260,E2 -1260} C_VEL
LIN {X 0,Y 594.239,Z 407.315,A -85,B 0,C 180,E1 -1260.678,E2 -1260.678} C_VEL
LIN {X 0,Y 594.239,Z 405.776,A -85,B 0,C 180,E1 -1262.033,E2 -1262.033} C_VEL
LIN {X 0,Y 594.226,Z 404.415,A -85,B 0,C 180,E1 -1262.712,E2 -1262.712} C_VEL
LIN {X 0,Y 594.289,Z 401.537,A -85,B 0,C 180,E1 -1263.729,E2 -1263.729} C_VEL
LIN {X 0,Y 594.241,Z 397.637,A -85,B 0,C 180,E1 -1264.749,E2 -1264.749} C_VEL
LIN {X 0,Y 594.299,Z 392.607,A -85,B 0,C 180,E1 -1265.769,E2 -1265.769} C_VEL
LIN {X 0,Y 594.317,Z 386.287,A -85,B 0,C 180,E1 -1266.791,E2 -1266.791} C_VEL
LIN {X 0,Y 594.347,Z 378.369,A -85,B 0,C 180,E1 -1267.816,E2 -1267.816} C_VEL
LIN {X 0,Y 594.381,Z 368.522,A -85,B 0,C 180,E1 -1268.842,E2 -1268.842} C_VEL
LIN {X 0,Y 594.426,Z 358.2,A -85,B 0,C 180,E1 -1269.7,E2 -1269.7} C_VEL
LIN {X 0,Y 594.503,Z 346.575,A -85,B 0,C 180,E1 -1270.472,E2 -1270.472} C_VEL
LIN {X 0,Y 594.569,Z 334.698,A -85,B 0,C 180,E1 -1271.088,E2 -1271.088} C_VEL
LIN {X 0,Y 594.56,Z 321.727,A -85,B 0,C 180,E1 -1271.593,E2 -1271.593} C_VEL
LIN {X 0,Y 594.607,Z 314.244,A -85,B 0,C 180,E1 -1271.814,E2 -1271.814} C_VEL
LIN {X 0,Y 593.984,Z 308.565,A -85,B 0,C 180,E1 -1271.962,E2 -1271.962} C_VEL
LIN {X 0,Y 588.823,Z 291.886,A -85,B 0,C 180,E1 -1272.327,E2 -1272.327} C_VEL
LIN {X 0,Y 587.844,Z 286.133,A -85,B 0,C 180,E1 -1272.416,E2 -1272.416} C_VEL
LIN {X 0,Y 587.782,Z 284.182,A -85,B 0,C 180,E1 -1272.441,E2 -1272.441} C_VEL
LIN {X 0,Y 587.72,Z 197.504,A -85,B 0,C 180,E1 -1273.507,E2 -1273.507} C_VEL
LIN {X 0,Y 587.391,Z 195.23,A -85,B 0,C 180,E1 -1273.558,E2 -1273.558} C_VEL
LIN {X 0,Y 587.49,Z 176.616,A -85,B 0,C 180,E1 -1276.149,E2 -1276.149} C_VEL
LIN {X 0,Y 587.61,Z 158.797,A -85,B 0,C 180,E1 -1278.659,E2 -1278.659} C_VEL
LIN {X 0,Y 587.754,Z 141.462,A -85,B 0,C 180,E1 -1281.143,E2 -1281.143} C_VEL
LIN {X 0,Y 587.864,Z 132.213,A -85,B 0,C 180,E1 -1282.493,E2 -1282.493} C_VEL
LIN {X 0,Y 587.323,Z 128.952,A -85,B 0,C 180,E1 -1283.024,E2 -1283.024} C_VEL
LIN {X 0,Y 587.333,Z 128.954,A -85,B 0,C 180,E1 -1285.517,E2 -1285.517} C_VEL
LIN {X 0,Y 587.307,Z 128.953,A -85,B 0,C 180,E1 -1287.82,E2 -1287.82} C_VEL
LIN {X 0,Y 587.325,Z 128.945,A -85,B 0,C 180,E1 -1290.507,E2 -1290.507} C_VEL
LIN {X 0,Y 587.336,Z 128.953,A -85,B 0,C 180,E1 -1293.397,E2 -1293.397} C_VEL
LIN {X 0,Y 587.292,Z 128.951,A -85,B 0,C 180,E1 -1295.9,E2 -1295.9} C_VEL
LIN {X 0,Y 587.323,Z 128.946,A -85,B 0,C 180,E1 -1298.48,E2 -1298.48} C_VEL
LIN {X 0,Y 587.337,Z 128.953,A -85,B 0,C 180,E1 -1301.157,E2 -1301.157} C_VEL
LIN {X 0,Y 587.316,Z 128.945,A -85,B 0,C 180,E1 -1304.112,E2 -1304.112} C_VEL
LIN {X 0,Y 587.313,Z 128.956,A -85,B 0,C 180,E1 -1306.993,E2 -1306.993} C_VEL
LIN {X 0,Y 587.314,Z 128.946,A -85,B 0,C 180,E1 -1309.745,E2 -1309.745} C_VEL
LIN {X 0,Y 587.347,Z 128.945,A -85,B 0,C 180,E1 -1312.392,E2 -1312.392} C_VEL
LIN {X 0,Y 587.345,Z 128.943,A -85,B 0,C 180,E1 -1315.653,E2 -1315.653} C_VEL
LIN {X 0,Y 587.344,Z 128.946,A -85,B 0,C 180,E1 -1318.231,E2 -1318.231} C_VEL
LIN {X 0,Y 587.352,Z 128.949,A -85,B 0,C 180,E1 -1320.867,E2 -1320.867} C_VEL
LIN {X 0,Y 587.343,Z 128.944,A -85,B 0,C 180,E1 -1323.823,E2 -1323.823} C_VEL
LIN {X 0,Y 587.327,Z 128.949,A -85,B 0,C 180,E1 -1325.992,E2 -1325.992} C_VEL
LIN {X 0,Y 587.358,Z 129.095,A -85,B 0,C 180,E1 -1327.123,E2 -1327.123} C_VEL
LIN {X 0,Y 587.868,Z 133.084,A -85,B 0,C 180,E1 -1327.692,E2 -1327.692} C_VEL
LIN {X 0,Y 587.707,Z 153.325,A -85,B 0,C 180,E1 -1330.437,E2 -1330.437} C_VEL
LIN {X 0,Y 587.678,Z 156.843,A -85,B 0,C 180,E1 -1330.909,E2 -1330.909} C_VEL
LIN {X 0,Y 588.579,Z 161.903,A -85,B 0,C 180,E1 -1331.016,E2 -1331.016} C_VEL
LIN {X 0,Y 588.295,Z 320.741,A -85,B 0,C 180,E1 -1333.022,E2 -1333.022} C_VEL
LIN {X 0,Y 588.222,Z 335.116,A -85,B 0,C 180,E1 -1333.317,E2 -1333.317} C_VEL
LIN {X 0,Y 588.074,Z 350.526,A -85,B 0,C 180,E1 -1333.778,E2 -1333.778} C_VEL
LIN {X 0,Y 587.991,Z 363.779,A -85,B 0,C 180,E1 -1334.31,E2 -1334.31} C_VEL
LIN {X 0,Y 587.834,Z 377.842,A -85,B 0,C 180,E1 -1335.016,E2 -1335.016} C_VEL
LIN {X 0,Y 587.725,Z 391.197,A -85,B 0,C 180,E1 -1335.84,E2 -1335.84} C_VEL
LIN {X 0,Y 587.582,Z 404.741,A -85,B 0,C 180,E1 -1336.864,E2 -1336.864} C_VEL
LIN {X 0,Y 587.455,Z 416.26,A -85,B 0,C 180,E1 -1337.914,E2 -1337.914} C_VEL
LIN {X 0,Y 587.352,Z 426.011,A -85,B 0,C 180,E1 -1338.962,E2 -1338.962} C_VEL
LIN {X 0,Y 587.311,Z 435.543,A -85,B 0,C 180,E1 -1340.181,E2 -1340.181} C_VEL
LIN {X 0,Y 587.268,Z 443.452,A -85,B 0,C 180,E1 -1341.396,E2 -1341.396} C_VEL
LIN {X 0,Y 587.217,Z 450.88,A -85,B 0,C 180,E1 -1342.78,E2 -1342.78} C_VEL
LIN {X 0,Y 587.227,Z 456.772,A -85,B 0,C 180,E1 -1344.16,E2 -1344.16} C_VEL
LIN {X 0,Y 587.134,Z 460.248,A -85,B 0,C 180,E1 -1345.193,E2 -1345.193} C_VEL
LIN {X 0,Y 587.179,Z 463.801,A -85,B 0,C 180,E1 -1346.568,E2 -1346.568} C_VEL
LIN {X 0,Y 587.14,Z 466.134,A -85,B 0,C 180,E1 -1347.941,E2 -1347.941} C_VEL
LIN {X 0,Y 587.135,Z 467.312,A -85,B 0,C 180,E1 -1349.313,E2 -1349.313} C_VEL
LIN {X 0,Y 587.136,Z 467.345,A -85,B 0,C 180,E1 -1350.685,E2 -1350.685} C_VEL
LIN {X 0,Y 587.14,Z 466.238,A -85,B 0,C 180,E1 -1352.057,E2 -1352.057} C_VEL
LIN {X 0,Y 587.181,Z 463.993,A -85,B 0,C 180,E1 -1353.43,E2 -1353.43} C_VEL
LIN {X 0,Y 587.134,Z 460.531,A -85,B 0,C 180,E1 -1354.806,E2 -1354.806} C_VEL
LIN {X 0,Y 587.183,Z 455.777,A -85,B 0,C 180,E1 -1356.183,E2 -1356.183} C_VEL
LIN {X 0,Y 587.215,Z 451.309,A -85,B 0,C 180,E1 -1357.218,E2 -1357.218} C_VEL
LIN {X 0,Y 587.265,Z 443.987,A -85,B 0,C 180,E1 -1358.602,E2 -1358.602} C_VEL
LIN {X 0,Y 587.305,Z 436.196,A -85,B 0,C 180,E1 -1359.817,E2 -1359.817} C_VEL
LIN {X 0,Y 587.383,Z 425.822,A -85,B 0,C 180,E1 -1361.15,E2 -1361.15} C_VEL
LIN {X 0,Y 587.491,Z 415.413,A -85,B 0,C 180,E1 -1362.258,E2 -1362.258} C_VEL
LIN {X 0,Y 587.613,Z 403.727,A -85,B 0,C 180,E1 -1363.31,E2 -1363.31} C_VEL
LIN {X 0,Y 587.763,Z 390.475,A -85,B 0,C 180,E1 -1364.299,E2 -1364.299} C_VEL
LIN {X 0,Y 587.831,Z 377.899,A -85,B 0,C 180,E1 -1365.071,E2 -1365.071} C_VEL
LIN {X 0,Y 587.995,Z 363.842,A -85,B 0,C 180,E1 -1365.777,E2 -1365.777} C_VEL
LIN {X 0,Y 588.132,Z 348.015,A -85,B 0,C 180,E1 -1366.397,E2 -1366.397} C_VEL
LIN {X 0,Y 588.233,Z 333.491,A -85,B 0,C 180,E1 -1366.812,E2 -1366.812} C_VEL
LIN {X 0,Y 588.293,Z 318.77,A -85,B 0,C 180,E1 -1367.1,E2 -1367.1} C_VEL
LIN {X 0,Y 588.464,Z 160.688,A -85,B 0,C 180,E1 -1369.094,E2 -1369.094} C_VEL
LIN {X 0,Y 587.7,Z 156.848,A -85,B 0,C 180,E1 -1369.18,E2 -1369.18} C_VEL
LIN {X 0,Y 587.867,Z 136.455,A -85,B 0,C 180,E1 -1371.936,E2 -1371.936} C_VEL
LIN {X 0,Y 587.795,Z 131.369,A -85,B 0,C 180,E1 -1372.636,E2 -1372.636} C_VEL
LIN {X 0,Y 587.325,Z 128.952,A -85,B 0,C 180,E1 -1372.998,E2 -1372.998} C_VEL
LIN {X 0,Y 587.335,Z 128.954,A -85,B 0,C 180,E1 -1375.515,E2 -1375.515} C_VEL
LIN {X 0,Y 587.345,Z 128.948,A -85,B 0,C 180,E1 -1377.817,E2 -1377.817} C_VEL
LIN {X 0,Y 587.338,Z 128.944,A -85,B 0,C 180,E1 -1380.51,E2 -1380.51} C_VEL
LIN {X 0,Y 587.338,Z 128.947,A -85,B 0,C 180,E1 -1383.111,E2 -1383.111} C_VEL
LIN {X 0,Y 587.351,Z 128.944,A -85,B 0,C 180,E1 -1385.894,E2 -1385.894} C_VEL
LIN {X 0,Y 587.327,Z 128.944,A -85,B 0,C 180,E1 -1388.478,E2 -1388.478} C_VEL
LIN {X 0,Y 587.332,Z 128.948,A -85,B 0,C 180,E1 -1391.156,E2 -1391.156} C_VEL
LIN {X 0,Y 587.328,Z 128.944,A -85,B 0,C 180,E1 -1394.113,E2 -1394.113} C_VEL
LIN {X 0,Y 587.308,Z 128.952,A -85,B 0,C 180,E1 -1396.993,E2 -1396.993} C_VEL
LIN {X 0,Y 587.313,Z 128.948,A -85,B 0,C 180,E1 -1399.745,E2 -1399.745} C_VEL
LIN {X 0,Y 587.338,Z 128.943,A -85,B 0,C 180,E1 -1402.392,E2 -1402.392} C_VEL
LIN {X 0,Y 587.345,Z 128.948,A -85,B 0,C 180,E1 -1404.945,E2 -1404.945} C_VEL
LIN {X 0,Y 587.332,Z 128.949,A -85,B 0,C 180,E1 -1407.42,E2 -1407.42} C_VEL
LIN {X 0,Y 587.339,Z 128.942,A -85,B 0,C 180,E1 -1409.83,E2 -1409.83} C_VEL
LIN {X 0,Y 587.342,Z 128.943,A -85,B 0,C 180,E1 -1412.306,E2 -1412.306} C_VEL
LIN {X 0,Y 587.327,Z 128.946,A -85,B 0,C 180,E1 -1414.483,E2 -1414.483} C_VEL
LIN {X 0,Y 587.31,Z 128.955,A -85,B 0,C 180,E1 -1417.13,E2 -1417.13} C_VEL
LIN {X 0,Y 587.325,Z 128.944,A -85,B 0,C 180,E1 -1419.695,E2 -1419.695} C_VEL
LIN {X 0,Y 587.349,Z 128.945,A -85,B 0,C 180,E1 -1422.594,E2 -1422.594} C_VEL
LIN {X 0,Y 587.354,Z 128.94,A -85,B 0,C 180,E1 -1425.739,E2 -1425.739} C_VEL
LIN {X 0,Y 587.352,Z 128.951,A -85,B 0,C 180,E1 -1428.858,E2 -1428.858} C_VEL
LIN {X 0,Y 587.361,Z 128.94,A -85,B 0,C 180,E1 -1431.745,E2 -1431.745} C_VEL
LIN {X 0,Y 587.355,Z 128.945,A -85,B 0,C 180,E1 -1434.507,E2 -1434.507} C_VEL
LIN {X 0,Y 587.374,Z 128.941,A -85,B 0,C 180,E1 -1437.257,E2 -1437.257} C_VEL
LIN {X 0,Y 587.368,Z 128.938,A -85,B 0,C 180,E1 -1440,E2 -1440} C_VEL
LIN {X 0,Y 587.373,Z 128.947,A -85,B 0,C 180,E1 -1442.743,E2 -1442.743} C_VEL
LIN {X 0,Y 587.353,Z 128.94,A -85,B 0,C 180,E1 -1445.493,E2 -1445.493} C_VEL
LIN {X 0,Y 587.361,Z 128.943,A -85,B 0,C 180,E1 -1448.255,E2 -1448.255} C_VEL
LIN {X 0,Y 587.351,Z 128.942,A -85,B 0,C 180,E1 -1451.141,E2 -1451.141} C_VEL
LIN {X 0,Y 587.354,Z 128.945,A -85,B 0,C 180,E1 -1454.261,E2 -1454.261} C_VEL
LIN {X 0,Y 587.35,Z 128.941,A -85,B 0,C 180,E1 -1457.406,E2 -1457.406} C_VEL
LIN {X 0,Y 587.326,Z 128.951,A -85,B 0,C 180,E1 -1460.305,E2 -1460.305} C_VEL
LIN {X 0,Y 587.354,Z 128.94,A -85,B 0,C 180,E1 -1463.257,E2 -1463.257} C_VEL
LIN {X 0,Y 587.348,Z 128.948,A -85,B 0,C 180,E1 -1466.182,E2 -1466.182} C_VEL
LIN {X 0,Y 587.341,Z 128.942,A -85,B 0,C 180,E1 -1469.135,E2 -1469.135} C_VEL
LIN {X 0,Y 587.347,Z 128.945,A -85,B 0,C 180,E1 -1471.838,E2 -1471.838} C_VEL
LIN {X 0,Y 587.348,Z 128.95,A -85,B 0,C 180,E1 -1474.35,E2 -1474.35} C_VEL
LIN {X 0,Y 587.344,Z 128.944,A -85,B 0,C 180,E1 -1476.747,E2 -1476.747} C_VEL
LIN {X 0,Y 587.326,Z 128.943,A -85,B 0,C 180,E1 -1479.361,E2 -1479.361} C_VEL
LIN {X 0,Y 587.326,Z 128.952,A -85,B 0,C 180,E1 -1482.109,E2 -1482.109} C_VEL
LIN {X 0,Y 587.308,Z 128.947,A -85,B 0,C 180,E1 -1485.09,E2 -1485.09} C_VEL
LIN {X 0,Y 587.345,Z 128.951,A -85,B 0,C 180,E1 -1487.928,E2 -1487.928} C_VEL
LIN {X 0,Y 587.325,Z 128.944,A -85,B 0,C 180,E1 -1491.059,E2 -1491.059} C_VEL
LIN {X 0,Y 587.346,Z 128.943,A -85,B 0,C 180,E1 -1493.293,E2 -1493.293} C_VEL
LIN {X 0,Y 587.356,Z 128.948,A -85,B 0,C 180,E1 -1495.781,E2 -1495.781} C_VEL
LIN {X 0,Y 587.335,Z 128.949,A -85,B 0,C 180,E1 -1498.232,E2 -1498.232} C_VEL
LIN {X 0,Y 587.345,Z 128.945,A -85,B 0,C 180,E1 -1500.868,E2 -1500.868} C_VEL
LIN {X 0,Y 587.36,Z 129.054,A -85,B 0,C 180,E1 -1501.675,E2 -1501.675} C_VEL
LIN {X 0,Y 588.996,Z 135.397,A -85,B 0,C 180,E1 -1502.268,E2 -1502.268} C_VEL
LIN {X 0,Y 588.801,Z 164.992,A -85,B 0,C 180,E1 -1504.656,E2 -1504.656} C_VEL
LIN {X 0,Y 588.462,Z 200.952,A -85,B 0,C 180,E1 -1507.533,E2 -1507.533} C_VEL
LIN {X 0,Y 588.118,Z 238.179,A -85,B 0,C 180,E1 -1510.453,E2 -1510.453} C_VEL
LIN {X 0,Y 588.099,Z 243.125,A -85,B 0,C 180,E1 -1510.838,E2 -1510.838} C_VEL
LIN {X 0,Y 588.597,Z 248.836,A -85,B 0,C 180,E1 -1510.933,E2 -1510.933} C_VEL
LIN {X 0,Y 588.304,Z 412.3,A -85,B 0,C 180,E1 -1512.998,E2 -1512.998} C_VEL
LIN {X 0,Y 588.213,Z 427.746,A -85,B 0,C 180,E1 -1513.337,E2 -1513.337} C_VEL
LIN {X 0,Y 588.084,Z 443.071,A -85,B 0,C 180,E1 -1513.824,E2 -1513.824} C_VEL
LIN {X 0,Y 587.995,Z 456.789,A -85,B 0,C 180,E1 -1514.4,E2 -1514.4} C_VEL
LIN {X 0,Y 587.839,Z 470.258,A -85,B 0,C 180,E1 -1515.106,E2 -1515.106} C_VEL
LIN {X 0,Y 587.738,Z 483.129,A -85,B 0,C 180,E1 -1515.93,E2 -1515.93} C_VEL
LIN {X 0,Y 587.582,Z 495.299,A -85,B 0,C 180,E1 -1516.865,E2 -1516.865} C_VEL
LIN {X 0,Y 587.453,Z 506.758,A -85,B 0,C 180,E1 -1517.916,E2 -1517.916} C_VEL
LIN {X 0,Y 587.348,Z 516.399,A -85,B 0,C 180,E1 -1518.964,E2 -1518.964} C_VEL
LIN {X 0,Y 587.304,Z 525.864,A -85,B 0,C 180,E1 -1520.183,E2 -1520.183} C_VEL
LIN {X 0,Y 587.265,Z 533.738,A -85,B 0,C 180,E1 -1521.398,E2 -1521.398} C_VEL
LIN {X 0,Y 587.214,Z 541.094,A -85,B 0,C 180,E1 -1522.782,E2 -1522.782} C_VEL
LIN {X 0,Y 587.227,Z 546.927,A -85,B 0,C 180,E1 -1524.162,E2 -1524.162} C_VEL
LIN {X 0,Y 587.136,Z 550.387,A -85,B 0,C 180,E1 -1525.194,E2 -1525.194} C_VEL
LIN {X 0,Y 587.179,Z 553.89,A -85,B 0,C 180,E1 -1526.57,E2 -1526.57} C_VEL
LIN {X 0,Y 587.14,Z 556.194,A -85,B 0,C 180,E1 -1527.943,E2 -1527.943} C_VEL
LIN {X 0,Y 587.138,Z 557.35,A -85,B 0,C 180,E1 -1529.315,E2 -1529.315} C_VEL
LIN {X 0,Y 587.138,Z 557.349,A -85,B 0,C 180,E1 -1530.687,E2 -1530.687} C_VEL
LIN {X 0,Y 587.14,Z 556.191,A -85,B 0,C 180,E1 -1532.059,E2 -1532.059} C_VEL
LIN {X 0,Y 587.179,Z 553.885,A -85,B 0,C 180,E1 -1533.432,E2 -1533.432} C_VEL
LIN {X 0,Y 587.136,Z 550.382,A -85,B 0,C 180,E1 -1534.807,E2 -1534.807} C_VEL
LIN {X 0,Y 587.181,Z 545.605,A -85,B 0,C 180,E1 -1536.185,E2 -1536.185} C_VEL
LIN {X 0,Y 587.23,Z 539.42,A -85,B 0,C 180,E1 -1537.566,E2 -1537.566} C_VEL
LIN {X 0,Y 587.266,Z 531.645,A -85,B 0,C 180,E1 -1538.951,E2 -1538.951} C_VEL
LIN {X 0,Y 587.351,Z 523.364,A -85,B 0,C 180,E1 -1540.166,E2 -1540.166} C_VEL
LIN {X 0,Y 587.401,Z 513.388,A -85,B 0,C 180,E1 -1541.386,E2 -1541.386} C_VEL
LIN {X 0,Y 587.522,Z 503.182,A -85,B 0,C 180,E1 -1542.435,E2 -1542.435} C_VEL
LIN {X 0,Y 587.629,Z 491.008,A -85,B 0,C 180,E1 -1543.487,E2 -1543.487} C_VEL
LIN {X 0,Y 587.776,Z 478.045,A -85,B 0,C 180,E1 -1544.417,E2 -1544.417} C_VEL
LIN {X 0,Y 587.928,Z 463.852,A -85,B 0,C 180,E1 -1545.248,E2 -1545.248} C_VEL
LIN {X 0,Y 588.034,Z 449.778,A -85,B 0,C 180,E1 -1545.912,E2 -1545.912} C_VEL
LIN {X 0,Y 588.171,Z 435.279,A -85,B 0,C 180,E1 -1546.442,E2 -1546.442} C_VEL
LIN {X 0,Y 588.263,Z 419.487,A -85,B 0,C 180,E1 -1546.862,E2 -1546.862} C_VEL
LIN {X 0,Y 588.3,Z 403.619,A -85,B 0,C 180,E1 -1547.13,E2 -1547.13} C_VEL
LIN {X 0,Y 588.503,Z 246.091,A -85,B 0,C 180,E1 -1549.105,E2 -1549.105} C_VEL
LIN {X 0,Y 588.088,Z 242.844,A -85,B 0,C 180,E1 -1549.184,E2 -1549.184} C_VEL
LIN {X 0,Y 588.415,Z 207.908,A -85,B 0,C 180,E1 -1551.917,E2 -1551.917} C_VEL
LIN {X 0,Y 588.712,Z 170.913,A -85,B 0,C 180,E1 -1554.868,E2 -1554.868} C_VEL
LIN {X 0,Y 588.95,Z 143.601,A -85,B 0,C 180,E1 -1557.062,E2 -1557.062} C_VEL
LIN {X 0,Y 588.758,Z 133.866,A -85,B 0,C 180,E1 -1557.852,E2 -1557.852} C_VEL
LIN {X 0,Y 587.335,Z 128.952,A -85,B 0,C 180,E1 -1558.329,E2 -1558.329} C_VEL
LIN {X 0,Y 587.322,Z 128.947,A -85,B 0,C 180,E1 -1560.968,E2 -1560.968} C_VEL
LIN {X 0,Y 587.334,Z 128.948,A -85,B 0,C 180,E1 -1563.397,E2 -1563.397} C_VEL
LIN {X 0,Y 587.281,Z 128.959,A -85,B 0,C 180,E1 -1565.902,E2 -1565.902} C_VEL
LIN {X 0,Y 587.306,Z 128.949,A -85,B 0,C 180,E1 -1568.482,E2 -1568.482} C_VEL
LIN {X 0,Y 587.312,Z 128.951,A -85,B 0,C 180,E1 -1571.16,E2 -1571.16} C_VEL
LIN {X 0,Y 587.287,Z 128.951,A -85,B 0,C 180,E1 -1574.109,E2 -1574.109} C_VEL
LIN {X 0,Y 587.283,Z 128.956,A -85,B 0,C 180,E1 -1576.991,E2 -1576.991} C_VEL
LIN {X 0,Y 587.281,Z 128.951,A -85,B 0,C 180,E1 -1579.987,E2 -1579.987} C_VEL
LIN {X 0,Y 587.302,Z 128.95,A -85,B 0,C 180,E1 -1582.389,E2 -1582.389} C_VEL
LIN {X 0,Y 587.33,Z 128.946,A -85,B 0,C 180,E1 -1585.656,E2 -1585.656} C_VEL
LIN {X 0,Y 587.318,Z 128.949,A -85,B 0,C 180,E1 -1588.23,E2 -1588.23} C_VEL
LIN {X 0,Y 587.34,Z 128.952,A -85,B 0,C 180,E1 -1590.869,E2 -1590.869} C_VEL
LIN {X 0,Y 587.308,Z 128.95,A -85,B 0,C 180,E1 -1593.83,E2 -1593.83} C_VEL
LIN {X 0,Y 587.304,Z 128.957,A -85,B 0,C 180,E1 -1596.741,E2 -1596.741} C_VEL
LIN {X 0,Y 587.33,Z 129.017,A -85,B 0,C 180,E1 -1597.035,E2 -1597.035} C_VEL
LIN {X 0,Y 587.896,Z 133.146,A -85,B 0,C 180,E1 -1597.694,E2 -1597.694} C_VEL
LIN {X 0,Y 587.715,Z 151.804,A -85,B 0,C 180,E1 -1600.438,E2 -1600.438} C_VEL
LIN {X 0,Y 587.525,Z 172.159,A -85,B 0,C 180,E1 -1603.316,E2 -1603.316} C_VEL
LIN {X 0,Y 587.425,Z 191.413,A -85,B 0,C 180,E1 -1606.003,E2 -1606.003} C_VEL
LIN {X 0,Y 587.428,Z 195.571,A -85,B 0,C 180,E1 -1606.553,E2 -1606.553} C_VEL
LIN {X 0,Y 587.845,Z 200.933,A -85,B 0,C 180,E1 -1606.629,E2 -1606.629} C_VEL
LIN {X 0,Y 587.734,Z 303.387,A -85,B 0,C 180,E1 -1607.899,E2 -1607.899} C_VEL
LIN {X 0,Y 587.699,Z 316.682,A -85,B 0,C 180,E1 -1608.205,E2 -1608.205} C_VEL
LIN {X 0,Y 587.613,Z 329.269,A -85,B 0,C 180,E1 -1608.635,E2 -1608.635} C_VEL
LIN {X 0,Y 587.539,Z 340.276,A -85,B 0,C 180,E1 -1609.141,E2 -1609.141} C_VEL
LIN {X 0,Y 587.448,Z 352.038,A -85,B 0,C 180,E1 -1609.836,E2 -1609.836} C_VEL
LIN {X 0,Y 587.39,Z 362.551,A -85,B 0,C 180,E1 -1610.618,E2 -1610.618} C_VEL
LIN {X 0,Y 587.323,Z 371.152,A -85,B 0,C 180,E1 -1611.398,E2 -1611.398} C_VEL
LIN {X 0,Y 587.274,Z 379.078,A -85,B 0,C 180,E1 -1612.263,E2 -1612.263} C_VEL
LIN {X 0,Y 587.236,Z 385.647,A -85,B 0,C 180,E1 -1613.126,E2 -1613.126} C_VEL
LIN {X 0,Y 587.237,Z 392.118,A -85,B 0,C 180,E1 -1614.161,E2 -1614.161} C_VEL
LIN {X 0,Y 587.146,Z 397.258,A -85,B 0,C 180,E1 -1615.194,E2 -1615.194} C_VEL
LIN {X 0,Y 587.213,Z 401.248,A -85,B 0,C 180,E1 -1616.226,E2 -1616.226} C_VEL
LIN {X 0,Y 587.132,Z 404.196,A -85,B 0,C 180,E1 -1617.256,E2 -1617.256} C_VEL
LIN {X 0,Y 587.139,Z 405.626,A -85,B 0,C 180,E1 -1617.942,E2 -1617.942} C_VEL
LIN {X 0,Y 587.141,Z 407.254,A -85,B 0,C 180,E1 -1619.314,E2 -1619.314} C_VEL
LIN {X 0,Y 587.137,Z 407.496,A -85,B 0,C 180,E1 -1620,E2 -1620} C_VEL
LIN {X 0,Y 587.14,Z 407.315,A -85,B 0,C 180,E1 -1620.686,E2 -1620.686} C_VEL
LIN {X 0,Y 587.138,Z 405.774,A -85,B 0,C 180,E1 -1622.058,E2 -1622.058} C_VEL
LIN {X 0,Y 587.133,Z 404.414,A -85,B 0,C 180,E1 -1622.744,E2 -1622.744} C_VEL
LIN {X 0,Y 587.213,Z 401.535,A -85,B 0,C 180,E1 -1623.774,E2 -1623.774} C_VEL
LIN {X 0,Y 587.147,Z 397.635,A -85,B 0,C 180,E1 -1624.806,E2 -1624.806} C_VEL
LIN {X 0,Y 587.229,Z 392.605,A -85,B 0,C 180,E1 -1625.839,E2 -1625.839} C_VEL
LIN {X 0,Y 587.231,Z 386.283,A -85,B 0,C 180,E1 -1626.874,E2 -1626.874} C_VEL
LIN {X 0,Y 587.288,Z 378.364,A -85,B 0,C 180,E1 -1627.91,E2 -1627.91} C_VEL
LIN {X 0,Y 587.343,Z 368.515,A -85,B 0,C 180,E1 -1628.949,E2 -1628.949} C_VEL
LIN {X 0,Y 587.411,Z 358.194,A -85,B 0,C 180,E1 -1629.817,E2 -1629.817} C_VEL
LIN {X 0,Y 587.519,Z 346.564,A -85,B 0,C 180,E1 -1630.598,E2 -1630.598} C_VEL
LIN {X 0,Y 587.593,Z 335.597,A -85,B 0,C 180,E1 -1631.18,E2 -1631.18} C_VEL
LIN {X 0,Y 587.599,Z 323.055,A -85,B 0,C 180,E1 -1631.686,E2 -1631.686} C_VEL
LIN {X 0,Y 587.696,Z 309.982,A -85,B 0,C 180,E1 -1632.058,E2 -1632.058} C_VEL
LIN {X 0,Y 587.741,Z 297.664,A -85,B 0,C 180,E1 -1632.276,E2 -1632.276} C_VEL
LIN {X 0,Y 587.782,Z 284.182,A -85,B 0,C 180,E1 -1632.441,E2 -1632.441} C_VEL
LIN {X 0,Y 587.182,Z 278.371,A -85,B 0,C 180,E1 -1632.525,E2 -1632.525} C_VEL
LIN {X 0,Y 581.592,Z 259.673,A -85,B 0,C 180,E1 -1632.879,E2 -1632.879} C_VEL
LIN {X 0,Y 580.926,Z 253.863,A -85,B 0,C 180,E1 -1632.966,E2 -1632.966} C_VEL
LIN {X 0,Y 580.809,Z 198.128,A -85,B 0,C 180,E1 -1633.662,E2 -1633.662} C_VEL
LIN {X 0,Y 580.394,Z 195.226,A -85,B 0,C 180,E1 -1633.725,E2 -1633.725} C_VEL
LIN {X 0,Y 580.541,Z 174.066,A -85,B 0,C 180,E1 -1636.709,E2 -1636.709} C_VEL
LIN {X 0,Y 580.73,Z 154.78,A -85,B 0,C 180,E1 -1639.478,E2 -1639.478} C_VEL
LIN {X 0,Y 580.972,Z 134.838,A -85,B 0,C 180,E1 -1642.399,E2 -1642.399} C_VEL
LIN {X 0,Y 580.286,Z 129.83,A -85,B 0,C 180,E1 -1643.184,E2 -1643.184} C_VEL
LIN {X 0,Y 580.309,Z 129.824,A -85,B 0,C 180,E1 -1645.08,E2 -1645.08} C_VEL
LIN {X 0,Y 580.28,Z 129.824,A -85,B 0,C 180,E1 -1648.187,E2 -1648.187} C_VEL
LIN {X 0,Y 580.275,Z 129.824,A -85,B 0,C 180,E1 -1650.692,E2 -1650.692} C_VEL
LIN {X 0,Y 580.306,Z 129.829,A -85,B 0,C 180,E1 -1653.316,E2 -1653.316} C_VEL
LIN {X 0,Y 580.247,Z 129.83,A -85,B 0,C 180,E1 -1655.756,E2 -1655.756} C_VEL
LIN {X 0,Y 580.288,Z 129.822,A -85,B 0,C 180,E1 -1658.146,E2 -1658.146} C_VEL
LIN {X 0,Y 580.299,Z 129.824,A -85,B 0,C 180,E1 -1660.844,E2 -1660.844} C_VEL
LIN {X 0,Y 580.274,Z 129.824,A -85,B 0,C 180,E1 -1663.658,E2 -1663.658} C_VEL
LIN {X 0,Y 580.273,Z 129.827,A -85,B 0,C 180,E1 -1666.61,E2 -1666.61} C_VEL
LIN {X 0,Y 580.3,Z 129.826,A -85,B 0,C 180,E1 -1669.156,E2 -1669.156} C_VEL
LIN {X 0,Y 580.291,Z 129.822,A -85,B 0,C 180,E1 -1671.927,E2 -1671.927} C_VEL
LIN {X 0,Y 580.253,Z 129.831,A -85,B 0,C 180,E1 -1674.452,E2 -1674.452} C_VEL
LIN {X 0,Y 580.294,Z 129.828,A -85,B 0,C 180,E1 -1676.975,E2 -1676.975} C_VEL
LIN {X 0,Y 580.288,Z 129.823,A -85,B 0,C 180,E1 -1679.424,E2 -1679.424} C_VEL
LIN {X 0,Y 580.296,Z 129.824,A -85,B 0,C 180,E1 -1682.142,E2 -1682.142} C_VEL
LIN {X 0,Y 580.325,Z 129.82,A -85,B 0,C 180,E1 -1685.269,E2 -1685.269} C_VEL
LIN {X 0,Y 580.313,Z 129.962,A -85,B 0,C 180,E1 -1686.949,E2 -1686.949} C_VEL
LIN {X 0,Y 580.964,Z 134.438,A -85,B 0,C 180,E1 -1687.6,E2 -1687.6} C_VEL
LIN {X 0,Y 580.783,Z 153.33,A -85,B 0,C 180,E1 -1690.194,E2 -1690.194} C_VEL
LIN {X 0,Y 580.749,Z 156.926,A -85,B 0,C 180,E1 -1690.683,E2 -1690.683} C_VEL
LIN {X 0,Y 581.875,Z 162.666,A -85,B 0,C 180,E1 -1690.798,E2 -1690.798} C_VEL
LIN {X 0,Y 581.53,Z 320.485,A -85,B 0,C 180,E1 -1692.814,E2 -1692.814} C_VEL
LIN {X 0,Y 581.442,Z 333.732,A -85,B 0,C 180,E1 -1693.083,E2 -1693.083} C_VEL
LIN {X 0,Y 581.278,Z 349.265,A -85,B 0,C 180,E1 -1693.538,E2 -1693.538} C_VEL
LIN {X 0,Y 581.148,Z 363.788,A -85,B 0,C 180,E1 -1694.12,E2 -1694.12} C_VEL
LIN {X 0,Y 580.991,Z 376.231,A -85,B 0,C 180,E1 -1694.745,E2 -1694.745} C_VEL
LIN {X 0,Y 580.811,Z 388.276,A -85,B 0,C 180,E1 -1695.472,E2 -1695.472} C_VEL
LIN {X 0,Y 580.663,Z 401.559,A -85,B 0,C 180,E1 -1696.437,E2 -1696.437} C_VEL
LIN {X 0,Y 580.535,Z 412.689,A -85,B 0,C 180,E1 -1697.413,E2 -1697.413} C_VEL
LIN {X 0,Y 580.392,Z 422.937,A -85,B 0,C 180,E1 -1698.474,E2 -1698.474} C_VEL
LIN {X 0,Y 580.331,Z 431.638,A -85,B 0,C 180,E1 -1699.533,E2 -1699.533} C_VEL
LIN {X 0,Y 580.214,Z 440.251,A -85,B 0,C 180,E1 -1700.764,E2 -1700.764} C_VEL
LIN {X 0,Y 580.178,Z 447.392,A -85,B 0,C 180,E1 -1701.992,E2 -1701.992} C_VEL
LIN {X 0,Y 580.126,Z 454.08,A -85,B 0,C 180,E1 -1703.413,E2 -1703.413} C_VEL
LIN {X 0,Y 580.075,Z 459.16,A -85,B 0,C 180,E1 -1704.786,E2 -1704.786} C_VEL
LIN {X 0,Y 580.087,Z 462.161,A -85,B 0,C 180,E1 -1705.831,E2 -1705.831} C_VEL
LIN {X 0,Y 580.038,Z 465.111,A -85,B 0,C 180,E1 -1707.221,E2 -1707.221} C_VEL
LIN {X 0,Y 580.043,Z 466.882,A -85,B 0,C 180,E1 -1708.611,E2 -1708.611} C_VEL
LIN {X 0,Y 580.035,Z 467.496,A -85,B 0,C 180,E1 -1709.999,E2 -1709.999} C_VEL
LIN {X 0,Y 580.045,Z 466.958,A -85,B 0,C 180,E1 -1711.388,E2 -1711.388} C_VEL
LIN {X 0,Y 580.04,Z 465.264,A -85,B 0,C 180,E1 -1712.777,E2 -1712.777} C_VEL
LIN {X 0,Y 580.087,Z 462.391,A -85,B 0,C 180,E1 -1714.168,E2 -1714.168} C_VEL
LIN {X 0,Y 580.127,Z 458.329,A -85,B 0,C 180,E1 -1715.561,E2 -1715.561} C_VEL
LIN {X 0,Y 580.138,Z 452.922,A -85,B 0,C 180,E1 -1716.957,E2 -1716.957} C_VEL
LIN {X 0,Y 580.172,Z 445.983,A -85,B 0,C 180,E1 -1718.357,E2 -1718.357} C_VEL
LIN {X 0,Y 580.229,Z 438.554,A -85,B 0,C 180,E1 -1719.586,E2 -1719.586} C_VEL
LIN {X 0,Y 580.329,Z 429.821,A -85,B 0,C 180,E1 -1720.794,E2 -1720.794} C_VEL
LIN {X 0,Y 580.426,Z 418.946,A -85,B 0,C 180,E1 -1722.055,E2 -1722.055} C_VEL
LIN {X 0,Y 580.587,Z 407.852,A -85,B 0,C 180,E1 -1723.118,E2 -1723.118} C_VEL
LIN {X 0,Y 580.718,Z 396.926,A -85,B 0,C 180,E1 -1724.006,E2 -1724.006} C_VEL
LIN {X 0,Y 580.91,Z 385.347,A -85,B 0,C 180,E1 -1724.807,E2 -1724.807} C_VEL
LIN {X 0,Y 581.066,Z 371.31,A -85,B 0,C 180,E1 -1725.61,E2 -1725.61} C_VEL
LIN {X 0,Y 581.214,Z 357.561,A -85,B 0,C 180,E1 -1726.237,E2 -1726.237} C_VEL
LIN {X 0,Y 581.313,Z 344.436,A -85,B 0,C 180,E1 -1726.708,E2 -1726.708} C_VEL
LIN {X 0,Y 581.436,Z 331.04,A -85,B 0,C 180,E1 -1727.071,E2 -1727.071} C_VEL
LIN {X 0,Y 581.554,Z 316.529,A -85,B 0,C 180,E1 -1727.338,E2 -1727.338} C_VEL
LIN {X 0,Y 581.795,Z 161.938,A -85,B 0,C 180,E1 -1729.304,E2 -1729.304} C_VEL
LIN {X 0,Y 580.761,Z 156.911,A -85,B 0,C 180,E1 -1729.409,E2 -1729.409} C_VEL
LIN {X 0,Y 580.968,Z 137.8,A -85,B 0,C 180,E1 -1732.024,E2 -1732.024} C_VEL
LIN {X 0,Y 580.807,Z 132.407,A -85,B 0,C 180,E1 -1732.78,E2 -1732.78} C_VEL
LIN {X 0,Y 580.288,Z 129.83,A -85,B 0,C 180,E1 -1733.167,E2 -1733.167} C_VEL
LIN {X 0,Y 580.292,Z 129.828,A -85,B 0,C 180,E1 -1735.848,E2 -1735.848} C_VEL
LIN {X 0,Y 580.297,Z 129.822,A -85,B 0,C 180,E1 -1738.184,E2 -1738.184} C_VEL
LIN {X 0,Y 580.288,Z 129.823,A -85,B 0,C 180,E1 -1740.695,E2 -1740.695} C_VEL
LIN {X 0,Y 580.302,Z 129.827,A -85,B 0,C 180,E1 -1743.316,E2 -1743.316} C_VEL
LIN {X 0,Y 580.32,Z 129.822,A -85,B 0,C 180,E1 -1745.766,E2 -1745.766} C_VEL
LIN {X 0,Y 580.284,Z 129.822,A -85,B 0,C 180,E1 -1748.145,E2 -1748.145} C_VEL
LIN {X 0,Y 580.295,Z 129.82,A -85,B 0,C 180,E1 -1750.842,E2 -1750.842} C_VEL
LIN {X 0,Y 580.282,Z 129.826,A -85,B 0,C 180,E1 -1753.656,E2 -1753.656} C_VEL
LIN {X 0,Y 580.27,Z 129.825,A -85,B 0,C 180,E1 -1756.608,E2 -1756.608} C_VEL
LIN {X 0,Y 580.293,Z 129.829,A -85,B 0,C 180,E1 -1759.156,E2 -1759.156} C_VEL
LIN {X 0,Y 580.284,Z 129.822,A -85,B 0,C 180,E1 -1761.926,E2 -1761.926} C_VEL
LIN {X 0,Y 580.301,Z 129.82,A -85,B 0,C 180,E1 -1764.456,E2 -1764.456} C_VEL
LIN {X 0,Y 580.283,Z 129.828,A -85,B 0,C 180,E1 -1766.975,E2 -1766.975} C_VEL
LIN {X 0,Y 580.302,Z 129.822,A -85,B 0,C 180,E1 -1769.425,E2 -1769.425} C_VEL
LIN {X 0,Y 580.311,Z 129.818,A -85,B 0,C 180,E1 -1772.136,E2 -1772.136} C_VEL
LIN {X 0,Y 580.312,Z 129.823,A -85,B 0,C 180,E1 -1775.269,E2 -1775.269} C_VEL
LIN {X 0,Y 580.265,Z 129.824,A -85,B 0,C 180,E1 -1777.947,E2 -1777.947} C_VEL
LIN {X 0,Y 580.308,Z 129.827,A -85,B 0,C 180,E1 -1780.914,E2 -1780.914} C_VEL
LIN {X 0,Y 580.275,Z 129.823,A -85,B 0,C 180,E1 -1783.825,E2 -1783.825} C_VEL
LIN {X 0,Y 580.273,Z 129.829,A -85,B 0,C 180,E1 -1786.696,E2 -1786.696} C_VEL
LIN {X 0,Y 580.294,Z 129.821,A -85,B 0,C 180,E1 -1789.533,E2 -1789.533} C_VEL
LIN {X 0,Y 580.323,Z 129.819,A -85,B 0,C 180,E1 -1792.344,E2 -1792.344} C_VEL
LIN {X 0,Y 580.333,Z 129.819,A -85,B 0,C 180,E1 -1795.137,E2 -1795.137} C_VEL
LIN {X 0,Y 580.324,Z 129.817,A -85,B 0,C 180,E1 -1797.918,E2 -1797.918} C_VEL
LIN {X 0,Y 580.361,Z 129.82,A -85,B 0,C 180,E1 -1800.694,E2 -1800.694} C_VEL
LIN {X 0,Y 580.281,Z 129.822,A -85,B 0,C 180,E1 -1803.472,E2 -1803.472} C_VEL
LIN {X 0,Y 580.318,Z 129.816,A -85,B 0,C 180,E1 -1805.56,E2 -1805.56} C_VEL
LIN {X 0,Y 580.325,Z 129.821,A -85,B 0,C 180,E1 -1808.356,E2 -1808.356} C_VEL
LIN {X 0,Y 580.322,Z 129.817,A -85,B 0,C 180,E1 -1811.208,E2 -1811.208} C_VEL
LIN {X 0,Y 580.304,Z 129.824,A -85,B 0,C 180,E1 -1814.339,E2 -1814.339} C_VEL
LIN {X 0,Y 580.305,Z 129.821,A -85,B 0,C 180,E1 -1816.916,E2 -1816.916} C_VEL
LIN {X 0,Y 580.298,Z 129.819,A -85,B 0,C 180,E1 -1819.822,E2 -1819.822} C_VEL
LIN {X 0,Y 580.318,Z 129.82,A -85,B 0,C 180,E1 -1822.801,E2 -1822.801} C_VEL
LIN {X 0,Y 580.296,Z 129.82,A -85,B 0,C 180,E1 -1825.08,E2 -1825.08} C_VEL
LIN {X 0,Y 580.294,Z 129.829,A -85,B 0,C 180,E1 -1828.186,E2 -1828.186} C_VEL
LIN {X 0,Y 580.284,Z 129.825,A -85,B 0,C 180,E1 -1830.697,E2 -1830.697} C_VEL
LIN {X 0,Y 580.293,Z 129.82,A -85,B 0,C 180,E1 -1833.317,E2 -1833.317} C_VEL
LIN {X 0,Y 580.317,Z 129.82,A -85,B 0,C 180,E1 -1835.768,E2 -1835.768} C_VEL
LIN {X 0,Y 580.281,Z 129.831,A -85,B 0,C 180,E1 -1838.147,E2 -1838.147} C_VEL
LIN {X 0,Y 580.294,Z 129.818,A -85,B 0,C 180,E1 -1840.844,E2 -1840.844} C_VEL
LIN {X 0,Y 580.271,Z 129.826,A -85,B 0,C 180,E1 -1843.659,E2 -1843.659} C_VEL
LIN {X 0,Y 580.277,Z 129.825,A -85,B 0,C 180,E1 -1846.609,E2 -1846.609} C_VEL
LIN {X 0,Y 580.293,Z 129.821,A -85,B 0,C 180,E1 -1849.158,E2 -1849.158} C_VEL
LIN {X 0,Y 580.284,Z 129.831,A -85,B 0,C 180,E1 -1851.928,E2 -1851.928} C_VEL
LIN {X 0,Y 580.279,Z 129.824,A -85,B 0,C 180,E1 -1854.456,E2 -1854.456} C_VEL
LIN {X 0,Y 580.285,Z 129.822,A -85,B 0,C 180,E1 -1856.976,E2 -1856.976} C_VEL
LIN {X 0,Y 580.297,Z 129.825,A -85,B 0,C 180,E1 -1859.427,E2 -1859.427} C_VEL
LIN {X 0,Y 580.288,Z 129.877,A -85,B 0,C 180,E1 -1861.396,E2 -1861.396} C_VEL
LIN {X 0,Y 582.333,Z 137.379,A -85,B 0,C 180,E1 -1862.12,E2 -1862.12} C_VEL
LIN {X 0,Y 582.069,Z 167.393,A -85,B 0,C 180,E1 -1864.553,E2 -1864.553} C_VEL
LIN {X 0,Y 581.72,Z 197.695,A -85,B 0,C 180,E1 -1866.995,E2 -1866.995} C_VEL
LIN {X 0,Y 581.406,Z 230.035,A -85,B 0,C 180,E1 -1869.573,E2 -1869.573} C_VEL
LIN {X 0,Y 581.254,Z 243.132,A -85,B 0,C 180,E1 -1870.604,E2 -1870.604} C_VEL
LIN {X 0,Y 581.888,Z 248.564,A -85,B 0,C 180,E1 -1870.701,E2 -1870.701} C_VEL
LIN {X 0,Y 581.521,Z 412.072,A -85,B 0,C 180,E1 -1872.79,E2 -1872.79} C_VEL
LIN {X 0,Y 581.419,Z 427.745,A -85,B 0,C 180,E1 -1873.137,E2 -1873.137} C_VEL
LIN {X 0,Y 581.253,Z 443.069,A -85,B 0,C 180,E1 -1873.629,E2 -1873.629} C_VEL
LIN {X 0,Y 581.122,Z 456.792,A -85,B 0,C 180,E1 -1874.211,E2 -1874.211} C_VEL
LIN {X 0,Y 580.949,Z 470.261,A -85,B 0,C 180,E1 -1874.925,E2 -1874.925} C_VEL
LIN {X 0,Y 580.802,Z 483.494,A -85,B 0,C 180,E1 -1875.784,E2 -1875.784} C_VEL
LIN {X 0,Y 580.607,Z 495.301,A -85,B 0,C 180,E1 -1876.705,E2 -1876.705} C_VEL
LIN {X 0,Y 580.478,Z 506.758,A -85,B 0,C 180,E1 -1877.769,E2 -1877.769} C_VEL
LIN {X 0,Y 580.307,Z 517.455,A -85,B 0,C 180,E1 -1878.954,E2 -1878.954} C_VEL
LIN {X 0,Y 580.268,Z 525.865,A -85,B 0,C 180,E1 -1880.062,E2 -1880.062} C_VEL
LIN {X 0,Y 580.214,Z 533.739,A -85,B 0,C 180,E1 -1881.292,E2 -1881.292} C_VEL
LIN {X 0,Y 580.13,Z 541.094,A -85,B 0,C 180,E1 -1882.693,E2 -1882.693} C_VEL
LIN {X 0,Y 580.131,Z 546.927,A -85,B 0,C 180,E1 -1884.091,E2 -1884.091} C_VEL
LIN {X 0,Y 580.041,Z 550.387,A -85,B 0,C 180,E1 -1885.136,E2 -1885.136} C_VEL
LIN {X 0,Y 580.104,Z 553.89,A -85,B 0,C 180,E1 -1886.528,E2 -1886.528} C_VEL
LIN {X 0,Y 580.039,Z 556.193,A -85,B 0,C 180,E1 -1887.918,E2 -1887.918} C_VEL
LIN {X 0,Y 580.038,Z 557.35,A -85,B 0,C 180,E1 -1889.307,E2 -1889.307} C_VEL
LIN {X 0,Y 580.038,Z 557.349,A -85,B 0,C 180,E1 -1890.695,E2 -1890.695} C_VEL
LIN {X 0,Y 580.039,Z 556.19,A -85,B 0,C 180,E1 -1892.084,E2 -1892.084} C_VEL
LIN {X 0,Y 580.105,Z 553.885,A -85,B 0,C 180,E1 -1893.474,E2 -1893.474} C_VEL
LIN {X 0,Y 580.041,Z 550.382,A -85,B 0,C 180,E1 -1894.866,E2 -1894.866} C_VEL
LIN {X 0,Y 580.093,Z 545.605,A -85,B 0,C 180,E1 -1896.261,E2 -1896.261} C_VEL
LIN {X 0,Y 580.166,Z 539.419,A -85,B 0,C 180,E1 -1897.658,E2 -1897.658} C_VEL
LIN {X 0,Y 580.207,Z 531.644,A -85,B 0,C 180,E1 -1899.061,E2 -1899.061} C_VEL
LIN {X 0,Y 580.309,Z 523.363,A -85,B 0,C 180,E1 -1900.291,E2 -1900.291} C_VEL
LIN {X 0,Y 580.384,Z 513.388,A -85,B 0,C 180,E1 -1901.526,E2 -1901.526} C_VEL
LIN {X 0,Y 580.541,Z 503.181,A -85,B 0,C 180,E1 -1902.587,E2 -1902.587} C_VEL
LIN {X 0,Y 580.689,Z 491.009,A -85,B 0,C 180,E1 -1903.652,E2 -1903.652} C_VEL
LIN {X 0,Y 580.877,Z 477.516,A -85,B 0,C 180,E1 -1904.626,E2 -1904.626} C_VEL
LIN {X 0,Y 581.055,Z 463.855,A -85,B 0,C 180,E1 -1905.433,E2 -1905.433} C_VEL
LIN {X 0,Y 581.194,Z 449.779,A -85,B 0,C 180,E1 -1906.104,E2 -1906.104} C_VEL
LIN {X 0,Y 581.359,Z 435.28,A -85,B 0,C 180,E1 -1906.641,E2 -1906.641} C_VEL
LIN {X 0,Y 581.476,Z 419.46,A -85,B 0,C 180,E1 -1907.066,E2 -1907.066} C_VEL
LIN {X 0,Y 581.531,Z 403.996,A -85,B 0,C 180,E1 -1907.331,E2 -1907.331} C_VEL
LIN {X 0,Y 581.903,Z 248.128,A -85,B 0,C 180,E1 -1909.305,E2 -1909.305} C_VEL
LIN {X 0,Y 581.285,Z 243.11,A -85,B 0,C 180,E1 -1909.397,E2 -1909.397} C_VEL
LIN {X 0,Y 581.631,Z 207.908,A -85,B 0,C 180,E1 -1912.186,E2 -1912.186} C_VEL
LIN {X 0,Y 582.041,Z 171.743,A -85,B 0,C 180,E1 -1915.095,E2 -1915.095} C_VEL
LIN {X 0,Y 582.256,Z 141.956,A -85,B 0,C 180,E1 -1917.484,E2 -1917.484} C_VEL
LIN {X 0,Y 582.037,Z 135.901,A -85,B 0,C 180,E1 -1917.986,E2 -1917.986} C_VEL
LIN {X 0,Y 580.301,Z 129.826,A -85,B 0,C 180,E1 -1918.581,E2 -1918.581} C_VEL
LIN {X 0,Y 580.269,Z 129.828,A -85,B 0,C 180,E1 -1921.387,E2 -1921.387} C_VEL
LIN {X 0,Y 580.311,Z 129.829,A -85,B 0,C 180,E1 -1923.856,E2 -1923.856} C_VEL
LIN {X 0,Y 580.284,Z 129.826,A -85,B 0,C 180,E1 -1927.27,E2 -1927.27} C_VEL
LIN {X 0,Y 580.276,Z 129.825,A -85,B 0,C 180,E1 -1930.269,E2 -1930.269} C_VEL
LIN {X 0,Y 580.248,Z 129.828,A -85,B 0,C 180,E1 -1932.71,E2 -1932.71} C_VEL
LIN {X 0,Y 580.248,Z 129.833,A -85,B 0,C 180,E1 -1935.612,E2 -1935.612} C_VEL
LIN {X 0,Y 580.23,Z 129.83,A -85,B 0,C 180,E1 -1938.227,E2 -1938.227} C_VEL
LIN {X 0,Y 580.256,Z 129.833,A -85,B 0,C 180,E1 -1940.963,E2 -1940.963} C_VEL
LIN {X 0,Y 580.232,Z 129.832,A -85,B 0,C 180,E1 -1943.594,E2 -1943.594} C_VEL
LIN {X 0,Y 580.268,Z 129.826,A -85,B 0,C 180,E1 -1946.142,E2 -1946.142} C_VEL
LIN {X 0,Y 580.255,Z 129.834,A -85,B 0,C 180,E1 -1948.613,E2 -1948.613} C_VEL
LIN {X 0,Y 580.279,Z 129.83,A -85,B 0,C 180,E1 -1951.023,E2 -1951.023} C_VEL
LIN {X 0,Y 580.267,Z 129.828,A -85,B 0,C 180,E1 -1953.672,E2 -1953.672} C_VEL
LIN {X 0,Y 580.254,Z 129.836,A -85,B 0,C 180,E1 -1956.441,E2 -1956.441} C_VEL
LIN {X 0,Y 580.3,Z 129.95,A -85,B 0,C 180,E1 -1956.798,E2 -1956.798} C_VEL
LIN {X 0,Y 581.106,Z 134.949,A -85,B 0,C 180,E1 -1957.606,E2 -1957.606} C_VEL
LIN {X 0,Y 580.785,Z 154.303,A -85,B 0,C 180,E1 -1960.524,E2 -1960.524} C_VEL
LIN {X 0,Y 580.542,Z 173.435,A -85,B 0,C 180,E1 -1963.291,E2 -1963.291} C_VEL
LIN {X 0,Y 580.415,Z 193.791,A -85,B 0,C 180,E1 -1966.164,E2 -1966.164} C_VEL
LIN {X 0,Y 580.425,Z 195.617,A -85,B 0,C 180,E1 -1966.387,E2 -1966.387} C_VEL
LIN {X 0,Y 580.96,Z 200.978,A -85,B 0,C 180,E1 -1966.467,E2 -1966.467} C_VEL
LIN {X 0,Y 580.809,Z 303.417,A -85,B 0,C 180,E1 -1967.753,E2 -1967.753} C_VEL
LIN {X 0,Y 580.771,Z 316.701,A -85,B 0,C 180,E1 -1968.062,E2 -1968.062} C_VEL
LIN {X 0,Y 580.677,Z 328.857,A -85,B 0,C 180,E1 -1968.481,E2 -1968.481} C_VEL
LIN {X 0,Y 580.549,Z 340.289,A -85,B 0,C 180,E1 -1969.008,E2 -1969.008} C_VEL
LIN {X 0,Y 580.429,Z 352.043,A -85,B 0,C 180,E1 -1969.712,E2 -1969.712} C_VEL
LIN {X 0,Y 580.341,Z 362.56,A -85,B 0,C 180,E1 -1970.503,E2 -1970.503} C_VEL
LIN {X 0,Y 580.272,Z 371.158,A -85,B 0,C 180,E1 -1971.292,E2 -1971.292} C_VEL
LIN {X 0,Y 580.222,Z 379.083,A -85,B 0,C 180,E1 -1972.168,E2 -1972.168} C_VEL
LIN {X 0,Y 580.169,Z 386.784,A -85,B 0,C 180,E1 -1973.21,E2 -1973.21} C_VEL
LIN {X 0,Y 580.139,Z 393.945,A -85,B 0,C 180,E1 -1974.439,E2 -1974.439} C_VEL
LIN {X 0,Y 580.108,Z 398.689,A -85,B 0,C 180,E1 -1975.484,E2 -1975.484} C_VEL
LIN {X 0,Y 580.123,Z 402.322,A -85,B 0,C 180,E1 -1976.527,E2 -1976.527} C_VEL
LIN {X 0,Y 580.043,Z 404.198,A -85,B 0,C 180,E1 -1977.222,E2 -1977.222} C_VEL
LIN {X 0,Y 580.038,Z 405.626,A -85,B 0,C 180,E1 -1977.917,E2 -1977.917} C_VEL
LIN {X 0,Y 580.041,Z 407.255,A -85,B 0,C 180,E1 -1979.306,E2 -1979.306} C_VEL
LIN {X 0,Y 580.038,Z 407.496,A -85,B 0,C 180,E1 -1980,E2 -1980} C_VEL
LIN {X 0,Y 580.04,Z 407.315,A -85,B 0,C 180,E1 -1980.694,E2 -1980.694} C_VEL
LIN {X 0,Y 580.037,Z 405.773,A -85,B 0,C 180,E1 -1982.083,E2 -1982.083} C_VEL
LIN {X 0,Y 580.044,Z 404.412,A -85,B 0,C 180,E1 -1982.778,E2 -1982.778} C_VEL
LIN {X 0,Y 580.11,Z 401.533,A -85,B 0,C 180,E1 -1983.821,E2 -1983.821} C_VEL
LIN {X 0,Y 580.053,Z 397.632,A -85,B 0,C 180,E1 -1984.865,E2 -1984.865} C_VEL
LIN {X 0,Y 580.162,Z 392.603,A -85,B 0,C 180,E1 -1985.91,E2 -1985.91} C_VEL
